IF doFrgVentilator THEN
    gStatusAnlage.Aktor[AKTOR_VENTILATOR] := STATUS_AKTIV;
ELSE
    gStatusAnlage.Aktor[AKTOR_VENTILATOR] := STATUS_NICHT_AKTIV;
END_IF;

aoFuVentilator := gAktoren.rVentilatorSollwert;

(*
===============================================================================
 LUFTAUFBEREITER
===============================================================================
 Direkte Ansteuerung
 Analoge Leistungsvorgabe analog zum Heizregister-Prinzip:
   - digitale Freigabe
   - analoger Sollwert
-------------------------------------------------------------------------------
*)

gStatusAnlage.LuftaufberTyp := gBetriebsparameter.Luftaufbereitung.Typ;


IF gAktoren.xFrgLuftaufbereiter THEN
    IF gAlarmBetriebLuftaufber THEN
        gStatusAnlage.Aktor[AKTOR_LUFTAUFBER] := STATUS_STOERUNG;
    ELSIF diBetriebLuftaufber THEN
        gStatusAnlage.Aktor[AKTOR_LUFTAUFBER] := STATUS_AKTIV;
    ELSE
        gStatusAnlage.Aktor[AKTOR_LUFTAUFBER] := STATUS_BEREIT;
    END_IF;
ELSE
    IF gAlarmBetriebLuftaufber THEN
        gStatusAnlage.Aktor[AKTOR_LUFTAUFBER] := STATUS_STOERUNG;
    ELSE
        gStatusAnlage.Aktor[AKTOR_LUFTAUFBER] := STATUS_NICHT_AKTIV;
    END_IF;
END_IF;

doFrgLuftaufber := gAktoren.xFrgLuftaufbereiter;
aoLeistVorgLuftaufber := gAktoren.rLuftaufbereiterSollwert;

(*
===============================================================================
 ABLUFTVENTILATOR
===============================================================================
 Direkte Ansteuerung
-------------------------------------------------------------------------------
*)

IF gAktoren.xFrgAbluftventilator THEN
    gStatusAnlage.Aktor[AKTOR_ABLUFTVENTILATOR] := STATUS_AKTIV;
ELSE
    gStatusAnlage.Aktor[AKTOR_ABLUFTVENTILATOR] := STATUS_NICHT_AKTIV;
END_IF;


doFrgAbluftventilator := gAktoren.xFrgAbluftventilator;
END_PROGRAM

PROGRAM HmiMappingCyclic
  VAR
    rt_Box_Aus : R_TRIG;
    rt_Box_Dauer : R_TRIG;
    rt_Box_Intervall : R_TRIG;
    rt_Box_Nachtr : R_TRIG;
    rt_Box_Stocktemp : R_TRIG;
    rt_Luftaufb_Auto : R_TRIG;
    rt_Luftaufb_Dauer : R_TRIG;
    rt_Luftaufb_Aus : R_TRIG;
    TOF_UmschBoxAktuell : TOF;  (* gemeinsam für Block A/B (schließen sich aus) *)
    TOF_UmschBox1 : TOF;  (* Block C (Einzelbox) *)
    xUmschSelAktuell : BOOL;
    xUmschSelBox1 : BOOL;
    lastBoxIndex : USINT;
    uIdx : USINT;
    firstStep : BOOL;
    xBox1BelegtLuefter : BOOL;
    xBox2BelegtLuefter : BOOL;
    TOF_Umsch : ARRAY[1..2] OF TOF;  (* eigener Hintergrund-Timer je Box *)
    xUmschTrig : ARRAY[1..2] OF BOOL;  (* Start-/Nachtrigger (Puls) je Box *)
    xZielAus : ARRAY[1..2] OF BOOL;  (* gewaehlte, noch nicht uebernommene Betriebsart *)
    xZielDauer : ARRAY[1..2] OF BOOL;
    xZielIntervall : ARRAY[1..2] OF BOOL;
    xZielNachtr : ARRAY[1..2] OF BOOL;
    xZielStocktemp : ARRAY[1..2] OF BOOL;
    xInitUmsch : BOOL := TRUE;
  END_VAR

(*
================================================================================
 File        : HMIMappingCyclic.st
 Project     : CControl_Lite
 Controller  : Schneider / EcoStruxure Machine Expert HVAC
 Author      : RIG Automation
 Created     : 2026-03-19
 Version     : V0.01
 Description :
    Zyklische Übergabe von Ein-/Ausgängen und aufbereiteten Messwerten an die HMI.

    Dieses Programm trennt bewusst zwischen:
      - Hardware-/Prozessabbild
      - interner Programmlogik
      - Visualisierungsdaten

    Die HMI liest ausschließlich die hier beschriebenen HMI-Variablen.
    Dadurch bleibt die Visualisierung von der eigentlichen I/O-Anbindung entkoppelt.

================================================================================
 Change History
--------------------------------------------------------------------------------
 Version | Date       | Author          | Description
--------------------------------------------------------------------------------
 V0.01   | 2026-03-19 | RIG Automation  | Initialerstellung HMI-Mapping für
                                        | digitale/analoge Ein- und Ausgänge
================================================================================
*)

(*
===============================================================================
 HMI-DATEN ZYKLISCH AKTUALISIEREN
-------------------------------------------------------------------------------
 Alle für die Visualisierung relevanten Ein- und Ausgangswerte werden in
 sprechende HMI-Variablen kopiert.
===============================================================================
*)
(*
---------------------------------------------------------------------------
Allgemein
---------------------------------------------------------------------------
*)
Konfig_SoftwareVersionPLC := gPlcSwVersion;
Konfig_idNameSteuerung := gPlcKonfigId;
gBetriebsparameter.Allgemein.StandortHoehe := Par_Anlage_Standorthoehe;


(*
---------------------------------------------------------------------------
Standard-Filterzeiten
---------------------------------------------------------------------------
*)
gBetriebsparameter.Sensoren.FilterzeitFrischluft := Sensoren_FilterzeitFrischluft;
gBetriebsparameter.Sensoren.FilterzeitAbluft := Sensoren_FilterzeitAbluft;
gBetriebsparameter.Sensoren.FilterzeitTrockenluft := Sensoren_FilterzeitTrockenluft;
gBetriebsparameter.Sensoren.FilterzeitStocktemp := Sensoren_FilterzeitStocktemp;

(*
---------------------------------------------------------------------------
Messbereiche Frischluft
---------------------------------------------------------------------------
*)
gBetriebsparameter.Sensoren.FrischlTempMessberMin := Sensoren_FrischlTempMessberMin;
gBetriebsparameter.Sensoren.FrischlTempMessberMax := Sensoren_FrischlTempMessberMax;
gBetriebsparameter.Sensoren.FrischlFeuchtMessberMin := Sensoren_FrischlFeuchteMessberMin;
gBetriebsparameter.Sensoren.FrischlFeuchtMessberMax := Sensoren_FrischlFeuchteMessberMax;

(*
---------------------------------------------------------------------------
Messbereiche Abluft
---------------------------------------------------------------------------
*)
gBetriebsparameter.Sensoren.AbluftTempMessberMin := Sensoren_AbluftTempMessberMin;
gBetriebsparameter.Sensoren.AbluftTempMessberMax := Sensoren_AbluftTempMessberMax;
gBetriebsparameter.Sensoren.AbluftFeuchtMessberMin := Sensoren_AbluftFeuchtMessberMin;
gBetriebsparameter.Sensoren.AbluftFeuchtMessberMax := Sensoren_AbluftFeuchtMessberMax;

(*
---------------------------------------------------------------------------
Messbereiche Trockenluft
---------------------------------------------------------------------------
*)
gBetriebsparameter.Sensoren.TrockenlTempMessberMin := Sensoren_TrockenlTempMessberMin;
gBetriebsparameter.Sensoren.TrockenlTempMessberMax := Sensoren_TrockenlTempMessberMax;
gBetriebsparameter.Sensoren.TrockenlFeuchtMessberMin := Sensoren_TrockenlFeuchtMessberMin;
gBetriebsparameter.Sensoren.TrockenlFeuchtMessberMax := Sensoren_TrockenlFeuchtMessberMax;

(*
---------------------------------------------------------------------------
Messbereiche Stocktemperatur
---------------------------------------------------------------------------
*)
gBetriebsparameter.Sensoren.StocktempMessberMin := Sensoren_StockTempMessberMin;
gBetriebsparameter.Sensoren.StocktempMessberMax := Sensoren_StockTempMessberMax;

(*
---------------------------------------------------------------------------
Sensor-Offsets
---------------------------------------------------------------------------
*)
gBetriebsparameter.Sensoren.OffsetFrischluftTemp := Sensoren_OffsetFrischluftTemp;
gBetriebsparameter.Sensoren.OffsetFrischluftFeuchte := Sensoren_OffsetFrischluftFeuchte;
gBetriebsparameter.Sensoren.OffsetAbluftBox1Temp := Sensoren_OffsetAbluftBox1Temp;
gBetriebsparameter.Sensoren.OffsetAbluftBox1Feuchte := Sensoren_OffsetAbluftBox1Feuchte;
gBetriebsparameter.Sensoren.OffsetAbluftBox2Temp := Sensoren_OffsetAbluftBox2Temp;
gBetriebsparameter.Sensoren.OffsetAbluftBox2Feuchte := Sensoren_OffsetAbluftBox2Feuchte;
gBetriebsparameter.Sensoren.OffsetTrockenluftTemp := Sensoren_OffsetTrockenluftTemp;
gBetriebsparameter.Sensoren.OffsetTrockenluftFeuchte := Sensoren_OffsetTrockenluftFeuchte;
gBetriebsparameter.Sensoren.OffsetStocktemp := Sensoren_OffsetStocktemp;

(*
---------------------------------------------------------------------------
Ausstattung / aktivierte Anlagenteile
---------------------------------------------------------------------------
Diese Werte sind vorläufige Defaultwerte und müssen später an die reale
Anlagenausstattung angepasst werden.
---------------------------------------------------------------------------
*)
gBetriebsparameter.Ausstattung.Box2 := Ausstattung_Box2;
gBetriebsparameter.Ausstattung.Abluftventilator := Ausstattung_Abluftventilator;
gBetriebsparameter.Ausstattung.SensorFrischluft := Ausstattung_SensorFrischluft;
gBetriebsparameter.Ausstattung.SensorAbluftBox1 := Ausstattung_SensorAbluftBox1;
gBetriebsparameter.Ausstattung.SensorAbluftBox2 := Ausstattung_SensorAbluftBox2;
gBetriebsparameter.Ausstattung.SensorTrockenluft := Ausstattung_SensorTrockenluft;
gBetriebsparameter.Ausstattung.SensorStocktemp := Ausstattung_SensorStocktemp;
gBetriebsparameter.Ausstattung.EndlagenVhdBoxenklappe1 := Ausstattung_EndlagenVhdBoxenklappe1;
gBetriebsparameter.Ausstattung.EndlagenVhdBoxenklappe2 := Ausstattung_EndlagenVhdBoxenklappe2;
gBetriebsparameter.Ausstattung.Luftaufbereiter := Ausstattung_Luftaufbereiter_Typ <> KEINER;

(*
---------------------------------------------------------------------------
Ventilator
---------------------------------------------------------------------------
*)
gBetriebsparameter.Ventilator.DrehzahlMin := Par_Ventilator_DrehzahlMin;
gBetriebsparameter.Ventilator.DrehzahlMax := Par_Ventilator_DrehzahlMax;
gBetriebsparameter.Ventilator.DrehzahlBeiAuskuehlphase := Par_Ventilator_DrehzahlBeiAuskuehlphase;
gBetriebsparameter.Ventilator.DrzUmschaltung := Par_Ventilator_DrzUmschaltung;
gBetriebsparameter.Ventilator.DrehzahlFixLuftaufbereiter := Par_Ventilator_DrehzahlFixLuftaufbereiter;
gBetriebsparameter.Ventilator.DrehzahlFixFrischluft := Par_Ventilator_DrehzahlFixFrischluft;
gBetriebsparameter.Ventilator.DrehzahlStrombegrenzung := Par_Ventilator_DrehzahlStrombegrenzung;
gBetriebsparameter.Ventilator.DrehzahlLeistungsreduziert := Par_Ventilator_DrehzahlLeistungsreduz;
gBetriebsparameter.Ventilator.ZeitRampeUp := Par_Ventilator_ZeitRampeUp;//[ms]
gBetriebsparameter.Ventilator.ZeitRampeDown := Par_Ventilator_ZeitRampeDown;//[ms]


(*
---------------------------------------------------------------------------
Luftaufbereitung
---------------------------------------------------------------------------
*)

//Allgemein
gBetriebsparameter.Luftaufbereitung.VerzWetterwechsel := Par_Luftaufbereitung_VerzWetterwechsel;
gBetriebsparameter.Luftaufbereitung.SaettigungFrischluftEin := Par_Luftaufbereitung_SaettigungFrischlEin;
gBetriebsparameter.Luftaufbereitung.Hysterese := Par_Luftaufbereitung_Hysterese;

//Betriebsarten
//--- Luftaufbereitung: Betriebsartenwahl (flankengesteuert, gegenseitig verriegelt) ---
rt_Luftaufb_Auto (CLK := Par_Luftaufbereitung_AutomatikbetriebEin);
rt_Luftaufb_Dauer(CLK := Par_Luftaufbereitung_DauerbetriebEin);
rt_Luftaufb_Aus  (CLK := Par_Luftaufbereitung_Aus);

IF rt_Luftaufb_Auto.Q THEN
	Par_Luftaufbereitung_DauerbetriebEin     := FALSE;
	Par_Luftaufbereitung_Aus                 := FALSE;
ELSIF rt_Luftaufb_Dauer.Q THEN
	Par_Luftaufbereitung_AutomatikbetriebEin := FALSE;
	Par_Luftaufbereitung_Aus                 := FALSE;
ELSIF rt_Luftaufb_Aus.Q THEN
	Par_Luftaufbereitung_AutomatikbetriebEin := FALSE;
	Par_Luftaufbereitung_DauerbetriebEin     := FALSE;
END_IF;

//Aufbereitete Anwahl an interne Betriebsparameter uebergeben
gBetriebsparameter.Luftaufbereitung.AutomatikbetriebEin := Par_Luftaufbereitung_AutomatikbetriebEin;
gBetriebsparameter.Luftaufbereitung.DauerbetriebEin     := Par_Luftaufbereitung_DauerbetriebEin;
gBetriebsparameter.Luftaufbereitung.Aus                 := Par_Luftaufbereitung_Aus;

//Spezifisch Heizregister
gBetriebsparameter.Luftaufbereitung.P := Par_Luftaufbereitung_P;
gBetriebsparameter.Luftaufbereitung.I := Par_Luftaufbereitung_I;
gBetriebsparameter.Luftaufbereitung.D := Par_Luftaufbereitung_D;
gBetriebsparameter.Luftaufbereitung.DrehzahlVorgabeMin := Par_Luftaufbereitung_DrehzahlVorgabeMin;
gBetriebsparameter.Luftaufbereitung.DrehzahlVorgabeMax := Par_Luftaufbereitung_DrehzahlVorgabeMax;
gBetriebsparameter.Luftaufbereitung.TempVorgabeSoll := Par_Luftaufbereitung_TempVorgabeSoll;
//Spezifisch Ofen
gBetriebsparameter.Luftaufbereitung.VerzBetriebsmeldung := Par_Luftaufbereitung_VerzBetriebsmeldung;
gBetriebsparameter.Luftaufbereitung.Auskuehlzeit := Par_Luftaufbereitung_Auskuehlzeit;
gBetriebsparameter.Luftaufbereitung.BetriebsmeldungVorh := Par_Luftaufbereitung_BetriebsmeldungVorh;

(*
---------------------------------------------------------------------------
Abluft
---------------------------------------------------------------------------
*)
gBetriebsparameter.Abluftventilator.FeuchteSoll := Par_Abluft_FeuchteSoll;
gBetriebsparameter.Abluftventilator.Hysterese := Par_Abluft_FeuchteHysterese;

(*
---------------------------------------------------------------------------
Schlechtwetter
---------------------------------------------------------------------------
*)

//======== Box 1 =========

//Sensortype 
gBetriebsparameter.SchlechtwetterBoxen[1].AuswahlSensorGrenzwert := Par_Schlechtwetter_Box1_Sensortype;
//Feuchte
gBetriebsparameter.SchlechtwetterBoxen[1].Stufe[1].MaterialfeuchteStufe := Par_Schlechtwetter_Box1_MaterialfeuchteStufe1;
gBetriebsparameter.SchlechtwetterBoxen[1].Stufe[2].MaterialfeuchteStufe := Par_Schlechtwetter_Box1_MaterialfeuchteStufe2;
gBetriebsparameter.SchlechtwetterBoxen[1].Stufe[3].MaterialfeuchteStufe := Par_Schlechtwetter_Box1_MaterialfeuchteStufe3;
gBetriebsparameter.SchlechtwetterBoxen[1].Stufe[4].MaterialfeuchteStufe := Par_Schlechtwetter_Box1_MaterialfeuchteStufe4;
gBetriebsparameter.SchlechtwetterBoxen[1].Stufe[5].MaterialfeuchteStufe := Par_Schlechtwetter_Box1_MaterialfeuchteStufe5;
gBetriebsparameter.SchlechtwetterBoxen[1].Stufe[6].MaterialfeuchteStufe := Par_Schlechtwetter_Box1_MaterialfeuchteStufe6;
//Saettigung
gBetriebsparameter.SchlechtwetterBoxen[1].Stufe[1].Saettigungsdefizit := Par_Schlechtwetter_Box1_Saettigungsdefizit1;
gBetriebsparameter.SchlechtwetterBoxen[1].Stufe[2].Saettigungsdefizit := Par_Schlechtwetter_Box1_Saettigungsdefizit2;
gBetriebsparameter.SchlechtwetterBoxen[1].Stufe[3].Saettigungsdefizit := Par_Schlechtwetter_Box1_Saettigungsdefizit3;
gBetriebsparameter.SchlechtwetterBoxen[1].Stufe[4].Saettigungsdefizit := Par_Schlechtwetter_Box1_Saettigungsdefizit4;
gBetriebsparameter.SchlechtwetterBoxen[1].Stufe[5].Saettigungsdefizit := Par_Schlechtwetter_Box1_Saettigungsdefizit5;
gBetriebsparameter.SchlechtwetterBoxen[1].Stufe[6].Saettigungsdefizit := Par_Schlechtwetter_Box1_Saettigungsdefizit6;
// Zeit Lauf
gBetriebsparameter.SchlechtwetterBoxen[1].Stufe[1].SchlechtwetterZeitLauf := Par_Schlechtwetter_Box1_ZeitLauf1;
gBetriebsparameter.SchlechtwetterBoxen[1].Stufe[2].SchlechtwetterZeitLauf := Par_Schlechtwetter_Box1_ZeitLauf2;
gBetriebsparameter.SchlechtwetterBoxen[1].Stufe[3].SchlechtwetterZeitLauf := Par_Schlechtwetter_Box1_ZeitLauf3;
gBetriebsparameter.SchlechtwetterBoxen[1].Stufe[4].SchlechtwetterZeitLauf := Par_Schlechtwetter_Box1_ZeitLauf4;
gBetriebsparameter.SchlechtwetterBoxen[1].Stufe[5].SchlechtwetterZeitLauf := Par_Schlechtwetter_Box1_ZeitLauf5;
gBetriebsparameter.SchlechtwetterBoxen[1].Stufe[6].SchlechtwetterZeitLauf := Par_Schlechtwetter_Box1_ZeitLauf6;
// Zeit Pause
gBetriebsparameter.SchlechtwetterBoxen[1].Stufe[1].SchlechtwetterZeitPause := Par_Schlechtwetter_Box1_ZeitPause1;
gBetriebsparameter.SchlechtwetterBoxen[1].Stufe[2].SchlechtwetterZeitPause := Par_Schlechtwetter_Box1_ZeitPause2;
gBetriebsparameter.SchlechtwetterBoxen[1].Stufe[3].SchlechtwetterZeitPause := Par_Schlechtwetter_Box1_ZeitPause3;
gBetriebsparameter.SchlechtwetterBoxen[1].Stufe[4].SchlechtwetterZeitPause := Par_Schlechtwetter_Box1_ZeitPause4;
gBetriebsparameter.SchlechtwetterBoxen[1].Stufe[5].SchlechtwetterZeitPause := Par_Schlechtwetter_Box1_ZeitPause5;
gBetriebsparameter.SchlechtwetterBoxen[1].Stufe[6].SchlechtwetterZeitPause := Par_Schlechtwetter_Box1_ZeitPause6;

gBetriebsparameter.SchlechtwetterBoxen[1].MaterialfeuchteIst := gBetriebsparameter.Boxen[1].AktuelleTrockengutFeuchte;
gBetriebsparameter.SchlechtwetterBoxen[1].HystereseGrenzwert := gBetriebsparameter.Luftaufbereitung.Hysterese;

//======== Box 2 =========

//Sensortype 
gBetriebsparameter.SchlechtwetterBoxen[2].AuswahlSensorGrenzwert := Par_Schlechtwetter_Box2_Sensortype;
//Feuchte
gBetriebsparameter.SchlechtwetterBoxen[2].Stufe[1].MaterialfeuchteStufe := Par_Schlechtwetter_Box2_MaterialfeuchteStufe1;
gBetriebsparameter.SchlechtwetterBoxen[2].Stufe[2].MaterialfeuchteStufe := Par_Schlechtwetter_Box2_MaterialfeuchteStufe2;
gBetriebsparameter.SchlechtwetterBoxen[2].Stufe[3].MaterialfeuchteStufe := Par_Schlechtwetter_Box2_MaterialfeuchteStufe3;
gBetriebsparameter.SchlechtwetterBoxen[2].Stufe[4].MaterialfeuchteStufe := Par_Schlechtwetter_Box2_MaterialfeuchteStufe4;
gBetriebsparameter.SchlechtwetterBoxen[2].Stufe[5].MaterialfeuchteStufe := Par_Schlechtwetter_Box2_MaterialfeuchteStufe5;
gBetriebsparameter.SchlechtwetterBoxen[2].Stufe[6].MaterialfeuchteStufe := Par_Schlechtwetter_Box2_MaterialfeuchteStufe6;
//Saettigung
gBetriebsparameter.SchlechtwetterBoxen[2].Stufe[1].Saettigungsdefizit := Par_Schlechtwetter_Box2_Saettigungsdefizit1;
gBetriebsparameter.SchlechtwetterBoxen[2].Stufe[2].Saettigungsdefizit := Par_Schlechtwetter_Box2_Saettigungsdefizit2;
gBetriebsparameter.SchlechtwetterBoxen[2].Stufe[3].Saettigungsdefizit := Par_Schlechtwetter_Box2_Saettigungsdefizit3;
gBetriebsparameter.SchlechtwetterBoxen[2].Stufe[4].Saettigungsdefizit := Par_Schlechtwetter_Box2_Saettigungsdefizit4;
gBetriebsparameter.SchlechtwetterBoxen[2].Stufe[5].Saettigungsdefizit := Par_Schlechtwetter_Box2_Saettigungsdefizit5;
gBetriebsparameter.SchlechtwetterBoxen[2].Stufe[6].Saettigungsdefizit := Par_Schlechtwetter_Box2_Saettigungsdefizit6;
// Zeit Lauf
gBetriebsparameter.SchlechtwetterBoxen[2].Stufe[1].SchlechtwetterZeitLauf := Par_Schlechtwetter_Box2_ZeitLauf1;
gBetriebsparameter.SchlechtwetterBoxen[2].Stufe[2].SchlechtwetterZeitLauf := Par_Schlechtwetter_Box2_ZeitLauf2;
gBetriebsparameter.SchlechtwetterBoxen[2].Stufe[3].SchlechtwetterZeitLauf := Par_Schlechtwetter_Box2_ZeitLauf3;
gBetriebsparameter.SchlechtwetterBoxen[2].Stufe[4].SchlechtwetterZeitLauf := Par_Schlechtwetter_Box2_ZeitLauf4;
gBetriebsparameter.SchlechtwetterBoxen[2].Stufe[5].SchlechtwetterZeitLauf := Par_Schlechtwetter_Box2_ZeitLauf5;
gBetriebsparameter.SchlechtwetterBoxen[2].Stufe[6].SchlechtwetterZeitLauf := Par_Schlechtwetter_Box2_ZeitLauf6;
// Zeit Pause
gBetriebsparameter.SchlechtwetterBoxen[2].Stufe[1].SchlechtwetterZeitPause := Par_Schlechtwetter_Box2_ZeitPause1;
gBetriebsparameter.SchlechtwetterBoxen[2].Stufe[2].SchlechtwetterZeitPause := Par_Schlechtwetter_Box2_ZeitPause2;
gBetriebsparameter.SchlechtwetterBoxen[2].Stufe[3].SchlechtwetterZeitPause := Par_Schlechtwetter_Box2_ZeitPause3;
gBetriebsparameter.SchlechtwetterBoxen[2].Stufe[4].SchlechtwetterZeitPause := Par_Schlechtwetter_Box2_ZeitPause4;
gBetriebsparameter.SchlechtwetterBoxen[2].Stufe[5].SchlechtwetterZeitPause := Par_Schlechtwetter_Box2_ZeitPause5;
gBetriebsparameter.SchlechtwetterBoxen[2].Stufe[6].SchlechtwetterZeitPause := Par_Schlechtwetter_Box2_ZeitPause6;

gBetriebsparameter.SchlechtwetterBoxen[2].MaterialfeuchteIst := gBetriebsparameter.Boxen[2].AktuelleTrockengutFeuchte;
gBetriebsparameter.SchlechtwetterBoxen[2].HystereseGrenzwert := gBetriebsparameter.Luftaufbereitung.Hysterese;

(*
---------------------------------------------------------------------------
Klappen/Boxen
---------------------------------------------------------------------------
*)
gBetriebsparameter.KlappenBoxen[1].Laufzeit := Klappen_Boxen_Box1_Laufzeit;
gBetriebsparameter.KlappenBoxen[2].Laufzeit := Klappen_Boxen_Box2_Laufzeit;

(*
---------------------------------------------------------------------------
Luftaufbereitung Allgemein
---------------------------------------------------------------------------
*)
gBetriebsparameter.Luftaufbereitung.Typ := Ausstattung_Luftaufbereiter_Typ;

(*
---------------------------------------------------------------------------
Strombegrenzung
---------------------------------------------------------------------------
*)
gBetriebsparameter.Strombegrenzung.StartStd := Par_Strombegrenzung_StartMin;
gBetriebsparameter.Strombegrenzung.StartMin := Par_Strombegrenzung_StartStd;
gBetriebsparameter.Strombegrenzung.StoppStd := Par_Strombegrenzung_StoppMin;
gBetriebsparameter.Strombegrenzung.StoppMin := Par_Strombegrenzung_StoppStd;
(*
---------------------------------------------------------------------------
Tarifabschaltung
---------------------------------------------------------------------------
*)
gBetriebsparameter.Tarifabschaltung.Zeitfenster.StartStd := Par_Tarifabschaltung_Start_Std;
gBetriebsparameter.Tarifabschaltung.Zeitfenster.StartMin := Par_Tarifabschaltung_Start_Min;
gBetriebsparameter.Tarifabschaltung.Zeitfenster.StoppStd := Par_Tarifabschaltung_Stopp_Std;
gBetriebsparameter.Tarifabschaltung.Zeitfenster.StoppMin := Par_Tarifabschaltung_Stopp_Min;
gBetriebsparameter.Tarifabschaltung.VorlaufzeitAbschaltungLuftaufb := Par_Vorlaufzeit_Luftaufb_Tarifabschalt;

(*
---------------------------------------------------------------------------
Verzoegerungen (alle in ms) 
---------------------------------------------------------------------------
*)
gBetriebsparameter.Verzoegerungen.Fehler                    := Par_Verz_Fehler;
gBetriebsparameter.Verzoegerungen.Warnungen                 := Par_Verz_Warnungen;
gBetriebsparameter.Verzoegerungen.AenderungKlappenstellung  := Par_Verz_Aenderung_Klappenstellung;
gBetriebsparameter.Verzoegerungen.UmschaltungBetriebsartBox := Par_Verz_Umsch_Betriebsart_Box;


(*
-------------------------------------------------------------------------------
 Betriebsart / allgemeiner Zustand
-------------------------------------------------------------------------------
*)
HMI_TEST_diIoTestAktiv:= (gAktModus = IOTEST);

(*
-------------------------------------------------------------------------------
 Digitale Eingänge an HMI übergeben
-------------------------------------------------------------------------------
*)
HMI_IN_diBox1Offen  		:= diBox1Offen;
HMI_IN_diBox1Geschl  		:= diBox1Geschl;
HMI_IN_diBox2Offen  		:= diBox2Offen;
HMI_IN_diBox2Geschl 		:= diBox2Geschl;
HMI_IN_diBetriebLuftaufber 	:= diBetriebLuftaufber;
HMI_IN_diBetriebVentilator 	:= diBetriebVentilator;

(*
-------------------------------------------------------------------------------
 Analoge Eingänge an HMI übergeben
-------------------------------------------------------------------------------
 Es werden bereits skalierte Engineering-Werte an die HMI übergeben.
-------------------------------------------------------------------------------
*)
HMI_IN_aiFrischluftTemp       := gStatusAnlage.FrischluftTemperatur;
HMI_IN_aiFrischluftFeuchte    := gStatusAnlage.FrischluftFeuchte;
HMI_IN_aiAbluftBox1Temp       := gStatusAnlage.AbluftBox1Temp;
HMI_IN_aiAbluftBox1Feuchte    := gStatusAnlage.AbluftBox1Feuchte;
HMI_IN_aiTrockenluftTemp      := gStatusAnlage.TrockenluftTemperatur;
HMI_IN_aiTrockenluftFeuchte   := gStatusAnlage.TrockenluftFeuchte;
HMI_IN_aiAbluftBox2Temp       := gStatusAnlage.AbluftBox2Temp;
HMI_IN_aiAbluftBox2Feuchte    := gStatusAnlage.AbluftBox2Feuchte;
HMI_IN_aiStocktemp            := gStatusAnlage.StockTemperatur;


(*
-------------------------------------------------------------------------------
 Digitale Ausgänge an HMI übergeben
-------------------------------------------------------------------------------
 Hier werden die internen Soll-/Freigabesignale visualisiert.
-------------------------------------------------------------------------------
*)
HMI_IN_doFrgLuftaufber     		:= doFrgLuftaufber;
HMI_IN_doFrgBox1            	:= doFrgBox1;
HMI_IN_doFrgBox2           		:= doFrgBox2;
HMI_IN_doFrgAbluftvent	     	:= doFrgAbluftventilator;
HMI_IN_doFrgVentilator	     	:= doFrgVentilator;

(*
-------------------------------------------------------------------------------
 Analogausgänge an HMI übergeben
-------------------------------------------------------------------------------
 Die HMI erhält die Engineering-Sollwerte sowie optional die bereits
 skalierten Hardwarewerte.
-------------------------------------------------------------------------------
*)
HMI_IN_aoFuVentilator   	  := aoFuVentilator;
HMI_IN_aoLeistVorgLuftaufber  := aoLeistVorgLuftaufber;


(*
-------------------------------------------------------------------------------
 Berechnete Werte an HMI übergeben
-------------------------------------------------------------------------------
*)
HMI_IN_FrischlSaettigunsDefizit := gStatusAnlage.FrischluftSaettDefizit;
HMI_IN_TrockenluftSaettigunsDefizit := gStatusAnlage.TrockenluftSaettDefizit;

(*
-------------------------------------------------------------------------------
 I/O-Testdaten an HMI übergeben
-------------------------------------------------------------------------------
 So sieht man in der Visu sofort, ob Testbetrieb aktiv ist und welche
 Testwerte gerade anliegen.
-------------------------------------------------------------------------------
*)


(* PLC OUT - HMI IN *)

//digital
HMI_TEST_diBox1Offen     		:= gIoTest.DigitalIn.diBox1Offen;
HMI_TEST_diBox1Geschl  	 		:= gIoTest.DigitalIn.diBox1Geschl;
HMI_TEST_diBox2Offen   		 	:= gIoTest.DigitalIn.diBox2Offen;
HMI_TEST_diBox2Geschl    		:= gIoTest.DigitalIn.diBox2Geschl;
HMI_TEST_diBetriebLuftaufber  	:= gIoTest.DigitalIn.diBetriebLuftaufber;
HMI_TEST_diBetriebVentilator 	:= gIoTest.DigitalIn.diBetriebVentilator;

//analog
HMI_TEST_aiFrischluftTemp  		:= gIoTest.AnalogIn.aiFrischluftTemp;
HMI_TEST_aiFrischluftFeuchte  	:= gIoTest.AnalogIn.aiFrischluftFeuchte;
HMI_TEST_aiAbluftBox1Temp     	:= gIoTest.AnalogIn.aiAbluftBox1Temp;
HMI_TEST_aiAbluftBox1Feuchte  	:= gIoTest.AnalogIn.aiAbluftBox1Feucht;
HMI_TEST_aiTrockenluftTemp 	  	:= gIoTest.AnalogIn.aiTrockenluftTemp;
HMI_TEST_aiTrockenluftFeuchte 	:= gIoTest.AnalogIn.aiTrockenluftFeucht;
HMI_TEST_aiAbluftBox2Temp  	  	:= gIoTest.AnalogIn.aiAbluftBox2Temp;
HMI_TEST_aiAbluftBox2Feuchte  	:= gIoTest.AnalogIn.aiAbluftBox2Feucht;
HMI_TEST_aiStocktemp   		  	:= gIoTest.AnalogIn.aiStocktemp;

(* HMI IN - PLC OUT *)

//digital
gIoTest.DigitalOut.doFrgLuftaufber			:= HMI_TEST_doFrgLuftaufber;
gIoTest.DigitalOut.doFrgBox1				:= HMI_TEST_doFrgBox1;
gIoTest.DigitalOut.doFrgBox2				:= HMI_TEST_doFrgBox2;
gIoTest.DigitalOut.doFrgAbluftventilator	:= HMI_TEST_doFrgAbluftventilator;
gIoTest.DigitalOut.doFrgVentilator			:= HMI_TEST_doFrgVentilator;

//analog
gIoTest.AnalogOut.aoFuVentilator			:= HMI_TEST_aoFuVentilator;
gIoTest.AnalogOut.aoLeistVorgLuftaufber 	:= HMI_TEST_aoLeistVorgLuftaufber;



(*
-------------------------------------------------------------------------------
 IO-MAPPING BOXEN 
-------------------------------------------------------------------------------
 Hier werden die Daten der Detailansichten der Boxen auf das allgemeine 
 PopUp geschrieben. Das allgemeine PopUp wird immer angezeigt wenn auf eine
 der Boxen geklickt wird. Die Daten der jeweiligen Box die ausgewählt wurde 
 werden dann auf dieses PopUp gemappet.
-------------------------------------------------------------------------------
*)

//======== Allgemein =========

gBetriebsparameter.Boxen[1].NameBox := Par_Box1_Name;
gBetriebsparameter.Boxen[2].NameBox := Par_Box2_Name;

//Trockengut
gBetriebsparameter.Boxen[1].Trockengut := Par_Boxen_1_Trockengut;
gBetriebsparameter.Boxen[2].Trockengut := Par_Boxen_2_Trockengut;

//Einstellung und Konfiguration Stellung Klappen
gBetriebsparameter.Boxen[1].StellungKlappe1 := Par_Box1_StellungKlappe1;
gBetriebsparameter.Boxen[1].StellungKlappe2 := Par_Box1_StellungKlappe2;
gBetriebsparameter.Boxen[2].StellungKlappe1 := Par_Box2_StellungKlappe1;
gBetriebsparameter.Boxen[2].StellungKlappe2 := Par_Box2_StellungKlappe2;

//Stocktemperatur
gBetriebsparameter.Boxen[1].StocktemperaturHysterese := Par_Stocktemperatur_Box1_Hysterese;
gBetriebsparameter.Boxen[2].StocktemperaturHysterese := Par_Stocktemperatur_Box2_Hysterese;

(*
-------------------------------------------------------------------------------
 Verriegelung Box-Betriebsarten (1 Luefter -> nur eine Box gleichzeitig)
 Belegt eine Box den Luefter durchgehend, wird bei der anderen Box
 Dauer-/Intervallbetrieb gesperrt (nur HMI-Hinweis).
-------------------------------------------------------------------------------
*)
// Reset
gStatusAnlage.Box[1].SperreDauerbetrieb     := FALSE;
gStatusAnlage.Box[1].SperreIntervallbetrieb := FALSE;
gStatusAnlage.Box[2].SperreDauerbetrieb     := FALSE;
gStatusAnlage.Box[2].SperreIntervallbetrieb := FALSE;

IF gBetriebsparameter.Ausstattung.Box2 THEN

    // "belegt den Luefter durchgehend" = Dauerbetrieb oder Stocktemperatur
    xBox1BelegtLuefter := gBetriebsparameter.Boxen[1].DauerbetriebEin
                          OR gBetriebsparameter.Boxen[1].StocktemperaturEin;
    xBox2BelegtLuefter := gBetriebsparameter.Boxen[2].DauerbetriebEin
                          OR gBetriebsparameter.Boxen[2].StocktemperaturEin;

    // Box 2 belegt den Luefter -> Box 1 sperren
    IF xBox2BelegtLuefter THEN
        gStatusAnlage.Box[1].SperreDauerbetrieb     := TRUE;
        gStatusAnlage.Box[1].SperreIntervallbetrieb := TRUE;
    ELSIF gBetriebsparameter.Boxen[2].IntervallbetriebEin THEN
        // Intervall der einen Box -> Dauerbetrieb der anderen wuerde stoeren
        gStatusAnlage.Box[1].SperreDauerbetrieb     := TRUE;
    END_IF;

    // Box 1 belegt den Luefter -> Box 2 sperren
    IF xBox1BelegtLuefter THEN
        gStatusAnlage.Box[2].SperreDauerbetrieb     := TRUE;
        gStatusAnlage.Box[2].SperreIntervallbetrieb := TRUE;
    ELSIF gBetriebsparameter.Boxen[1].IntervallbetriebEin THEN
        gStatusAnlage.Box[2].SperreDauerbetrieb     := TRUE;
    END_IF;

END_IF;

// --- HMI-Spiegel ---
HMI_IN_Box1_SperreDauerbetrieb     := gStatusAnlage.Box[1].SperreDauerbetrieb;
HMI_IN_Box1_SperreIntervallbetrieb := gStatusAnlage.Box[1].SperreIntervallbetrieb;
HMI_IN_Box2_SperreDauerbetrieb     := gStatusAnlage.Box[2].SperreDauerbetrieb;
HMI_IN_Box2_SperreIntervallbetrieb := gStatusAnlage.Box[2].SperreIntervallbetrieb;

// Aktuell-PopUp je nach angezeigter Box
IF HMI_OUT_Box_Aktuell_BoxIndex = BOX_2 THEN
    HMI_IN_Box_Aktuell_SperreDauerbetrieb     := gStatusAnlage.Box[2].SperreDauerbetrieb;
    HMI_IN_Box_Aktuell_SperreIntervallbetrieb := gStatusAnlage.Box[2].SperreIntervallbetrieb;
ELSE
    HMI_IN_Box_Aktuell_SperreDauerbetrieb     := gStatusAnlage.Box[1].SperreDauerbetrieb;
    HMI_IN_Box_Aktuell_SperreIntervallbetrieb := gStatusAnlage.Box[1].SperreIntervallbetrieb;
END_IF;

//======== Box 1 =========
HMI_IN_Box1_IconWitterung := gStatusAnlage.Box[1].IconWitterung;
HMI_IN_Box1_LaufRestzeitMinuten := gStatusAnlage.Box[1].LaufRestzeitMinuten;
HMI_IN_Box1_LaufRestzeitStunden := gStatusAnlage.Box[1].LaufRestzeitStunden;
HMI_IN_Box1_Status := TO_UINT(gStatusAnlage.Box[1].Status);
HMI_IN_Box1_TextIndexLaufzeit := gStatusAnlage.Box[1].TextIndexLaufzeit;
HMI_IN_Box1_TrockengutIcon := gStatusAnlage.Box[1].TrockengutIcon;
HMI_IN_Box1_AnzeigeLaufRestzeit := gStatusAnlage.Box[1].AnzeigeLaufRestzeit;

//TODO RIG: Noch zu verschalten
//HMI_IN_Box1_RestzeitUmschVerzBetriebsart

//======== Box 2 =========
HMI_IN_Box2_IconWitterung := gStatusAnlage.Box[2].IconWitterung;
HMI_IN_Box2_LaufRestzeitMinuten := gStatusAnlage.Box[2].LaufRestzeitMinuten;
HMI_IN_Box2_LaufRestzeitStunden := gStatusAnlage.Box[2].LaufRestzeitStunden;
HMI_IN_Box2_Status := TO_UINT(gStatusAnlage.Box[2].Status);
HMI_IN_Box2_TextIndexLaufzeit := gStatusAnlage.Box[2].TextIndexLaufzeit;
HMI_IN_Box2_TrockengutIcon := gStatusAnlage.Box[2].TrockengutIcon;
HMI_IN_Box2_AnzeigeLaufRestzeit := gStatusAnlage.Box[2].AnzeigeLaufRestzeit;

//TODO RIG: Noch zu verschalten
//HMI_IN_Box2_RestzeitUmschVerzBetriebsart

IF lastBoxIndex <> HMI_OUT_Box_Aktuell_BoxIndex THEN
	firstStep := TRUE;
	lastBoxIndex := HMI_OUT_Box_Aktuell_BoxIndex;
END_IF;

(*
-------------------------------------------------------------------------------
 Zusatzmeldung Anlagenstatus (vereinfacht fuer Lite) - nur Statustext
-------------------------------------------------------------------------------
*)
IF gAktModus = STILLSTAND THEN
    IF gAktoren.xLuftaufbNachlauf AND NOT gAktoren.xFrgLuftaufbereiter THEN
        HMI_Zusatzmeldung_Statustext := ZM_AUSKUEHLZEIT_WLO_AKTIV;      // Auskuehlung laeuft
    ELSIF gCmdAnlage.FehlerStopp THEN
        HMI_Zusatzmeldung_Statustext := ZM_STILLSTAND_FEHLERSTOPP;      // Fehler - kein Start
    ELSE
        HMI_Zusatzmeldung_Statustext := ZM_STILLSTAND_BEREIT;          // bereit
    END_IF;

ELSIF gAktModus = IOTEST THEN
    HMI_Zusatzmeldung_Statustext := ZM_STILLSTAND_IOTEST_NICHT_ABGE;    // I/O-Test aktiv

ELSE   // BETRIEB
    HMI_Zusatzmeldung_Restzeit 	:= 0;   //Kein Countdown
    HMI_Zusatzmeldung_Sanduhr 	:= 0;	//Keine Sanduhr
    IF gCmdAnlage.xTarifAbschaltung THEN
        HMI_Zusatzmeldung_Statustext := ZM_TARIFABSCHALTUNG_AKTIV;
    ELSIF gCmdAnlage.xTarifAbschaltungLuftaufb THEN
        HMI_Zusatzmeldung_Statustext := ZM_FRISCHLUFTB_VLZ_TARIF;
    ELSIF Strombegrenzung.StrombegrenzungEin THEN
        HMI_Zusatzmeldung_Statustext := ZM_STROMBEGRENZUNG_AKTIV;
    ELSIF (gStatusAnlage.Aktor[AKTOR_KLAPPE_BOX_1] = STATUS_IN_BEWEGUNG)
       OR (gStatusAnlage.Aktor[AKTOR_KLAPPE_BOX_2] = STATUS_IN_BEWEGUNG) THEN
        HMI_Zusatzmeldung_Statustext := ZM_KLAPPEN_WERDEN_UMGESCHALTET;
        HMI_Zusatzmeldung_Restzeit   := HMI_IN_Box_Aktuell_RestzeitUmschVerzBetriebsart;  
        HMI_Zusatzmeldung_Sanduhr := 1;
    ELSIF gAktoren.xLuftaufbNachlauf AND NOT gAktoren.xFrgLuftaufbereiter THEN
        HMI_Zusatzmeldung_Statustext := ZM_AUSKUEHLZEIT_WLO_AKTIV;
        HMI_Zusatzmeldung_Restzeit   := gAktoren.uRestAuskuehlzeitLuftaufb;   
    ELSE
        HMI_Zusatzmeldung_Statustext := ZM_FRISCHLUFTBETRIEB;
    END_IF;
END_IF;


//Box 1 auf Aktualfenster PopUp schreiben
IF HMI_OUT_Box_Aktuell_BoxIndex = BOX_1 THEN
	
	IF firstStep THEN
		HMI_OUT_Box_Aktuell_Aus                 := xZielAus[1];
		HMI_OUT_Box_Aktuell_DauerbetriebEin     := xZielDauer[1];
		HMI_OUT_Box_Aktuell_IntervallbetriebEIn := xZielIntervall[1];
		HMI_OUT_Box_Aktuell_NachtrocknungEin    := xZielNachtr[1];
		HMI_OUT_Box_Aktuell_StocktemperaturEin  := xZielStocktemp[1];
		HMI_OUT_Box_Aktuell_TrockengutfeuchteAktuell := gBetriebsparameter.Boxen[1].AktuelleTrockengutFeuchte;
		HMI_OUT_Box_Aktuell_StocktemperaturSoll := gBetriebsparameter.Boxen[1].StocktemperaturSoll;
		firstStep := FALSE;
	END_IF;
		
	//--- Gewaehlte Betriebsart als Ziel merken + Hintergrund-Timer starten ---
	IF rt_Box_Aus.Q OR rt_Box_Dauer.Q OR rt_Box_Intervall.Q OR rt_Box_Nachtr.Q OR rt_Box_Stocktemp.Q THEN
		xZielAus[1]       := HMI_OUT_Box_Aktuell_Aus;
		xZielDauer[1]     := HMI_OUT_Box_Aktuell_DauerbetriebEin;
		xZielIntervall[1] := HMI_OUT_Box_Aktuell_IntervallbetriebEIn;
		xZielNachtr[1]    := HMI_OUT_Box_Aktuell_NachtrocknungEin;
		xZielStocktemp[1] := HMI_OUT_Box_Aktuell_StocktemperaturEin;
		xUmschTrig[1]     := TRUE;
	END_IF;
	
	HMI_IN_Box_Aktuell_RestzeitUmschVerzBetriebsart := TO_UINT(gBetriebsparameter.Verzoegerungen.UmschaltungBetriebsartBox - TOF_Umsch[1].ET);
	//Aktuelle Trockengutfeuchte - Einstellung aus HMI
	gBetriebsparameter.Boxen[1].AktuelleTrockengutFeuchte := HMI_OUT_Box_Aktuell_TrockengutfeuchteAktuell;
	gBetriebsparameter.Boxen[1].StocktemperaturSoll := 	HMI_OUT_Box_Aktuell_StocktemperaturSoll;
	
	
	//PLC -> HMI
	HMI_IN_Box_Aktuell_Name := gBetriebsparameter.Boxen[1].NameBox;
	HMI_IN_Box_Aktuell_Temp := gStatusAnlage.AbluftBox1Temp;
	HMI_IN_Box_Aktuell_Feucht := gStatusAnlage.AbluftBox1Feuchte;	
	HMI_IN_Box_Aktuell_TrockengutIcon := gStatusAnlage.Box[1].TrockengutIcon;
	HMI_IN_Box_Aktuell_LaufRestzeitMinuten := gStatusAnlage.Box[1].LaufRestzeitMinuten;
	HMI_IN_Box_Aktuell_LaufRestzeitStunden := gStatusAnlage.Box[1].LaufRestzeitStunden;
	HMI_IN_Box_Aktuell_IconWitterung := gStatusAnlage.Box[1].IconWitterung;
	HMI_IN_Box_Aktuell_Status := TO_INT(gStatusAnlage.Box[1].Status);
	HMI_IN_Box_Aktuell_TextIndexLaufzeit := gStatusAnlage.Box[1].TextIndexLaufzeit;
	HMI_IN_Box_Aktuell_AnzeigeLaufRestzeit := gStatusAnlage.Box[1].AnzeigeLaufRestzeit;
	
	
//Box 2 auf Aktualfenster-PopUp schreiben
ELSIF HMI_OUT_Box_Aktuell_BoxIndex = BOX_2 THEN

	IF firstStep THEN
		HMI_OUT_Box_Aktuell_Aus                 := xZielAus[2];
		HMI_OUT_Box_Aktuell_DauerbetriebEin     := xZielDauer[2];
		HMI_OUT_Box_Aktuell_IntervallbetriebEIn := xZielIntervall[2];
		HMI_OUT_Box_Aktuell_NachtrocknungEin    := xZielNachtr[2];
		HMI_OUT_Box_Aktuell_StocktemperaturEin  := xZielStocktemp[2];
		HMI_OUT_Box_Aktuell_TrockengutfeuchteAktuell := gBetriebsparameter.Boxen[2].AktuelleTrockengutFeuchte;
		HMI_OUT_Box_Aktuell_StocktemperaturSoll := gBetriebsparameter.Boxen[2].StocktemperaturSoll;
		firstStep := FALSE;
	END_IF;

	//HMI -> PLC	
	//--- Gewaehlte Betriebsart als Ziel merken + Hintergrund-Timer starten ---
	IF rt_Box_Aus.Q OR rt_Box_Dauer.Q OR rt_Box_Intervall.Q OR rt_Box_Nachtr.Q OR rt_Box_Stocktemp.Q THEN
		xZielAus[2]       := HMI_OUT_Box_Aktuell_Aus;
		xZielDauer[2]     := HMI_OUT_Box_Aktuell_DauerbetriebEin;
		xZielIntervall[2] := HMI_OUT_Box_Aktuell_IntervallbetriebEIn;
		xZielNachtr[2]    := HMI_OUT_Box_Aktuell_NachtrocknungEin;
		xZielStocktemp[2] := HMI_OUT_Box_Aktuell_StocktemperaturEin;
		xUmschTrig[2]     := TRUE;
	END_IF;
	
	HMI_IN_Box_Aktuell_RestzeitUmschVerzBetriebsart := TO_UINT(gBetriebsparameter.Verzoegerungen.UmschaltungBetriebsartBox - TOF_Umsch[2].ET);
	//Aktuelle Trockengutfeuchte - Einstellung aus HMI
	gBetriebsparameter.Boxen[2].AktuelleTrockengutFeuchte := HMI_OUT_Box_Aktuell_TrockengutfeuchteAktuell;
	gBetriebsparameter.Boxen[2].StocktemperaturSoll := 	HMI_OUT_Box_Aktuell_StocktemperaturSoll;
		
	//PLC -> HMI
	HMI_IN_Box_Aktuell_Name := gBetriebsparameter.Boxen[2].NameBox;
	HMI_IN_Box_Aktuell_Temp := gStatusAnlage.AbluftBox2Temp;
	HMI_IN_Box_Aktuell_Feucht := gStatusAnlage.AbluftBox2Feuchte;	
	HMI_IN_Box_Aktuell_TrockengutIcon := gStatusAnlage.Box[2].TrockengutIcon;
	HMI_IN_Box_Aktuell_LaufRestzeitMinuten := gStatusAnlage.Box[2].LaufRestzeitMinuten;
	HMI_IN_Box_Aktuell_LaufRestzeitStunden := gStatusAnlage.Box[2].LaufRestzeitStunden;
	HMI_IN_Box_Aktuell_IconWitterung := gStatusAnlage.Box[2].IconWitterung;
	HMI_IN_Box_Aktuell_Status := TO_INT(gStatusAnlage.Box[2].Status);
	HMI_IN_Box_Aktuell_TextIndexLaufzeit := gStatusAnlage.Box[2].TextIndexLaufzeit;
	HMI_IN_Box_Aktuell_AnzeigeLaufRestzeit := gStatusAnlage.Box[2].AnzeigeLaufRestzeit;
	
ELSE 
	//nichts zu tun
END_IF;

IF (NOT gBetriebsparameter.Ausstattung.Box2) THEN
//--- Nur eine Box verfuegbar - Box 1 ist einzige Box : Betriebsartenwahl (flankengesteuert) ---
	firstStep := FALSE;
	rt_Box_Aus(CLK := HMI_OUT_Box1_Aus);
	rt_Box_Dauer(CLK := HMI_OUT_Box1_DauerbetriebEin);
	rt_Box_Intervall(CLK := HMI_OUT_Box1_IntervallbetriebEIn);
	rt_Box_Nachtr(CLK := HMI_OUT_Box1_NachtrocknungEin);
	rt_Box_Stocktemp(CLK := HMI_OUT_Box1_StocktemperaturEin);
	
	IF rt_Box_Aus.Q THEN
	    HMI_OUT_Box1_DauerbetriebEin     := FALSE;
	    HMI_OUT_Box1_IntervallbetriebEIn := FALSE;
	    HMI_OUT_Box1_NachtrocknungEin    := FALSE;
	    HMI_OUT_Box1_StocktemperaturEin  := FALSE;
	ELSIF rt_Box_Dauer.Q THEN
	    HMI_OUT_Box1_Aus                 := FALSE;
	    HMI_OUT_Box1_IntervallbetriebEIn := FALSE;
	    HMI_OUT_Box1_NachtrocknungEin    := FALSE;
	    HMI_OUT_Box1_StocktemperaturEin  := FALSE;
	ELSIF rt_Box_Intervall.Q THEN
	    HMI_OUT_Box1_Aus                 := FALSE;
	    HMI_OUT_Box1_DauerbetriebEin     := FALSE;
	    HMI_OUT_Box1_NachtrocknungEin    := FALSE;
	    HMI_OUT_Box1_StocktemperaturEin  := FALSE;
	ELSIF rt_Box_Nachtr.Q THEN
	    HMI_OUT_Box1_Aus                 := FALSE;
	    HMI_OUT_Box1_DauerbetriebEin     := FALSE;
	    HMI_OUT_Box1_IntervallbetriebEIn := FALSE;
	    HMI_OUT_Box1_StocktemperaturEin  := FALSE;
	ELSIF rt_Box_Stocktemp.Q THEN
	    HMI_OUT_Box1_Aus                 := FALSE;
	    HMI_OUT_Box1_DauerbetriebEin     := FALSE;
	    HMI_OUT_Box1_IntervallbetriebEIn := FALSE;
	    HMI_OUT_Box1_NachtrocknungEin 	 := FALSE;		
	END_IF;
	
	//--- Betriebsart verzögert übernehmen ---
	//--- Gewaehlte Betriebsart als Ziel merken + Hintergrund-Timer starten ---
	IF rt_Box_Aus.Q OR rt_Box_Dauer.Q OR rt_Box_Intervall.Q OR rt_Box_Nachtr.Q OR rt_Box_Stocktemp.Q THEN
		xZielAus[1]       := HMI_OUT_Box1_Aus;
		xZielDauer[1]     := HMI_OUT_Box1_DauerbetriebEin;
		xZielIntervall[1] := HMI_OUT_Box1_IntervallbetriebEIn;
		xZielNachtr[1]    := HMI_OUT_Box1_NachtrocknungEin;
		xZielStocktemp[1] := HMI_OUT_Box1_StocktemperaturEin;
		xUmschTrig[1]     := TRUE;
	END_IF;
	
	HMI_IN_Box1_RestzeitUmschVerzBetriebsart := TO_UINT(gBetriebsparameter.Verzoegerungen.UmschaltungBetriebsartBox - TOF_Umsch[1].ET);	
	
	//Aktuelle Trockengutfeuchte - Einstellung aus HMI
	gBetriebsparameter.Boxen[1].AktuelleTrockengutFeuchte := HMI_OUT_Box_Aktuell_TrockengutfeuchteAktuell;
	gBetriebsparameter.Boxen[1].StocktemperaturSoll := 	HMI_OUT_Box_Aktuell_StocktemperaturSoll;
	//Detailansicht Box 2
	
	//BOX 2 HIER EINFACH NUR GEH LOSSN!!! Wird in der VISU verwaltet!
	
END_IF;

//======================================================================
// Verzoegerte Betriebsart-Umschaltung (Hintergrund, eigener Timer je Box)
// - laeuft immer, auch wenn das Popup geschlossen ist
// - solange Timer laeuft bleibt die ALTE Betriebsart aktiv
// - erst nach Ablauf wird die neue Betriebsart uebernommen
//======================================================================
IF xInitUmsch THEN
	// Ziel = aktuell aktive Betriebsart -> kein Umschalten beim Anlauf
	FOR uIdx := 1 TO 2 DO
		xZielAus[uIdx]       := gBetriebsparameter.Boxen[uIdx].Aus;
		xZielDauer[uIdx]     := gBetriebsparameter.Boxen[uIdx].DauerbetriebEin;
		xZielIntervall[uIdx] := gBetriebsparameter.Boxen[uIdx].IntervallbetriebEin;
		xZielNachtr[uIdx]    := gBetriebsparameter.Boxen[uIdx].NachtrocknungEin;
		xZielStocktemp[uIdx] := gBetriebsparameter.Boxen[uIdx].StocktemperaturEin;
	END_FOR;
	xInitUmsch := FALSE;
END_IF;

FOR uIdx := 1 TO 2 DO
	TOF_Umsch[uIdx](IN := xUmschTrig[uIdx],
	                PT := gBetriebsparameter.Verzoegerungen.UmschaltungBetriebsartBox);
	xUmschTrig[uIdx] := FALSE;   // Trigger ist nur ein Puls (Timer haelt selbst nach)

	// Solange Timer laeuft (Q=TRUE) NICHT uebernehmen -> alte Betriebsart bleibt.
	// Nach Ablauf (Q=FALSE) neue Betriebsart uebernehmen.
	IF NOT TOF_Umsch[uIdx].Q THEN
		gBetriebsparameter.Boxen[uIdx].Aus                 := xZielAus[uIdx];
		gBetriebsparameter.Boxen[uIdx].DauerbetriebEin     := xZielDauer[uIdx];
		gBetriebsparameter.Boxen[uIdx].IntervallbetriebEin := xZielIntervall[uIdx];
		gBetriebsparameter.Boxen[uIdx].NachtrocknungEin    := xZielNachtr[uIdx];
		gBetriebsparameter.Boxen[uIdx].StocktemperaturEin  := xZielStocktemp[uIdx];
	END_IF;
END_FOR;

(*
-------------------------------------------------------------------------------
 SICHTBARKEITEN UND STATUS
-------------------------------------------------------------------------------
*)

//Lauf Restzeit einfach immer anzeigen
HMI_IN_Box1_AnzeigeLaufRestzeit := ICON_VISIBLE;
HMI_IN_Box2_AnzeigeLaufRestzeit := ICON_VISIBLE;

//Ventilator
IF gAlarmBetriebVentilator THEN 
	HMI_Ventilator1_FarbeIcon := ICON_ROT;
ELSIF gAktoren.xFrgVentilator THEN
	HMI_Ventilator1_FarbeIcon := ICON_GELB;
ELSE 
	HMI_Ventilator1_FarbeIcon := ICON_GRAU;
END_IF;

//Luftaufbereitung Icon
IF gBetriebsparameter.Ausstattung.Luftaufbereiter THEN 
	IF gAlarmBetriebLuftaufber THEN 
		Par_Luftaufbereitung_FarbeIcon := ICON_ROT;
	ELSIF gAktoren.xFrgLuftaufbereiter THEN
		Par_Luftaufbereitung_FarbeIcon := ICON_GELB;
	ELSE 
		Par_Luftaufbereitung_FarbeIcon := ICON_GRAU;
	END_IF;
ELSE 
	Par_Luftaufbereitung_FarbeIcon := ICON_HIDDEN;	
END_IF;

//Statusindex Textbox Luftaufbereiter PopUp
HMI_IN_LuftaufberStatusIndex := TO_USINT(gStatusAnlage.Aktor[AKTOR_LUFTAUFBER]);

//Abluftventilator
IF gBetriebsparameter.Ausstattung.Abluftventilator THEN 
	IF FALSE THEN //Abluftventilator hat keinen Alarm
		HMI_Abluft_FarbeIcon := ICON_ROT;
	ELSIF gAktoren.xFrgAbluftventilator THEN
		HMI_Abluft_FarbeIcon := ICON_GELB;
	ELSE 
		HMI_Abluft_FarbeIcon := ICON_GRAU;
	END_IF;
ELSE 
	HMI_Abluft_FarbeIcon := ICON_HIDDEN;	
END_IF;

// ===================== BOX 1 Status (Text fuer VISU) =====================
IF gCmdAnlage.Test THEN
    gStatusAnlage.Box[1].Status := STATUS_TESTBETRIEB;
ELSIF gBetriebsparameter.Boxen[1].Aus THEN
    gStatusAnlage.Box[1].Status := STATUS_STILLSTAND;
ELSIF gBetriebsparameter.Boxen[1].DauerbetriebEin THEN
    IF gStatusAnlage.Box[1].WetterIstSchlecht
       AND NOT (gBetriebsparameter.Ausstattung.Luftaufbereiter
                AND (gBetriebsparameter.Luftaufbereitung.Typ = HEIZREGISTER OR gBetriebsparameter.Luftaufbereitung.Typ = OFEN)
                AND (gBetriebsparameter.Luftaufbereitung.AutomatikbetriebEin OR gBetriebsparameter.Luftaufbereitung.DauerbetriebEin)) THEN
        IF gBetriebsparameter.Boxen[1].xBoxAktiv THEN
            gStatusAnlage.Box[1].Status := STATUS_SCHLECHTWETTER_LAUF;
        ELSE
            gStatusAnlage.Box[1].Status := STATUS_SCHLECHTWETTER_PAUSE;
        END_IF;
    ELSIF gBetriebsparameter.Boxen[1].xBoxAktiv THEN
        gStatusAnlage.Box[1].Status := STATUS_DAUERBETRIEB;
    ELSE
        gStatusAnlage.Box[1].Status := STATUS_DAUERBETRIEB_PAUSIERT;
    END_IF;
ELSIF gBetriebsparameter.Boxen[1].IntervallbetriebEin THEN
    IF gBetriebsparameter.Boxen[1].xBoxAktiv THEN
        gStatusAnlage.Box[1].Status := STATUS_INTERVALL_LAUF;
    ELSE
        gStatusAnlage.Box[1].Status := STATUS_INTERVALL_PAUSE;
    END_IF;
ELSIF gBetriebsparameter.Boxen[1].NachtrocknungEin THEN
    IF gBetriebsparameter.Boxen[1].xBoxAktiv THEN
        gStatusAnlage.Box[1].Status := STATUS_NACHTROCKNUNG_LAUF;
    ELSE
        gStatusAnlage.Box[1].Status := STATUS_NACHTROCKNUNG_PAUSE;
    END_IF;
ELSIF gBetriebsparameter.Boxen[1].StocktemperaturEin THEN
    IF gBetriebsparameter.Boxen[1].xBoxAktiv THEN
        gStatusAnlage.Box[1].Status := STATUS_STOCKTEMPERATUR_LAUF;       
    ELSE
        gStatusAnlage.Box[1].Status := STATUS_STOCKTEMPERATUR_PAUSE;
    END_IF;
ELSE
    gStatusAnlage.Box[1].Status := STATUS_STILLSTAND;
END_IF;

//BOX 2
// ===================== BOX 2 Status (Text fuer VISU) =====================
IF NOT gBetriebsparameter.Ausstattung.Box2 THEN
    gStatusAnlage.Box[2].Status := STATUS_NICHT_VERFUEGBAR;
ELSIF gCmdAnlage.Test THEN
    gStatusAnlage.Box[2].Status := STATUS_TESTBETRIEB;
ELSIF gBetriebsparameter.Boxen[2].Aus THEN
    gStatusAnlage.Box[2].Status := STATUS_STILLSTAND;
ELSIF gBetriebsparameter.Boxen[2].DauerbetriebEin THEN
    IF gStatusAnlage.Box[2].WetterIstSchlecht
       AND NOT (gBetriebsparameter.Ausstattung.Luftaufbereiter
                AND (gBetriebsparameter.Luftaufbereitung.Typ = HEIZREGISTER OR gBetriebsparameter.Luftaufbereitung.Typ = OFEN)
                AND (gBetriebsparameter.Luftaufbereitung.AutomatikbetriebEin OR gBetriebsparameter.Luftaufbereitung.DauerbetriebEin)) THEN
        IF gBetriebsparameter.Boxen[2].xBoxAktiv THEN
            gStatusAnlage.Box[2].Status := STATUS_SCHLECHTWETTER_LAUF;
        ELSE
            gStatusAnlage.Box[2].Status := STATUS_SCHLECHTWETTER_PAUSE;
        END_IF;
    ELSIF gBetriebsparameter.Boxen[2].xBoxAktiv THEN
        gStatusAnlage.Box[2].Status := STATUS_DAUERBETRIEB;
    ELSE
        gStatusAnlage.Box[2].Status := STATUS_DAUERBETRIEB_PAUSIERT;
    END_IF;
ELSIF gBetriebsparameter.Boxen[2].IntervallbetriebEin THEN
    IF gBetriebsparameter.Boxen[2].xBoxAktiv THEN
        gStatusAnlage.Box[2].Status := STATUS_INTERVALL_LAUF;
    ELSE
        gStatusAnlage.Box[2].Status := STATUS_INTERVALL_PAUSE;
    END_IF;
ELSIF gBetriebsparameter.Boxen[2].NachtrocknungEin THEN
    IF gBetriebsparameter.Boxen[2].xBoxAktiv THEN
        gStatusAnlage.Box[2].Status := STATUS_NACHTROCKNUNG_LAUF;
    ELSE
        gStatusAnlage.Box[2].Status := STATUS_NACHTROCKNUNG_PAUSE;
    END_IF;
ELSIF gBetriebsparameter.Boxen[2].StocktemperaturEin THEN
    IF gBetriebsparameter.Boxen[2].xBoxAktiv THEN
        gStatusAnlage.Box[2].Status := STATUS_STOCKTEMPERATUR_LAUF;
    ELSE
        gStatusAnlage.Box[2].Status := STATUS_STOCKTEMPERATUR_PAUSE;
    END_IF;
ELSE
    gStatusAnlage.Box[2].Status := STATUS_STILLSTAND;
END_IF;

(*
-------------------------------------------------------------------------------
 ALARME fuer Visu aufbereiten ARRAY -> UDINT Maske da Arrays nicht direkt
 an HMI gesendet werden koennen! 
-------------------------------------------------------------------------------
*)

//Reset Bitmasken vor Auswertung
HMI_IN_ALARM_WARNMASKE_1 := fcResetBitmask();
HMI_IN_ALARM_WARNMASKE_2 := fcResetBitmask();
HMI_IN_ALARM_STOERMASKE_1 := fcResetBitmask();
HMI_IN_ALARM_STOERMASKE_2 := fcResetBitmask();

//Array auf Bitmaske fuer HMI schreiben
FOR uIdx := 0 TO 31 DO
	//Erste Warnungsbitmaske [0.31]
	IF (gStatusAnlage.Alarm.ArrWarnung[uIdx]) THEN
		HMI_IN_ALARM_WARNMASKE_1:= fcSetBitInBitmask(Bitmask := HMI_IN_ALARM_WARNMASKE_1, BitNr:= uIdx);
	END_IF;
	//Zweite Warnungsbitmaske [32.63]
	IF (gStatusAnlage.Alarm.ArrWarnung[uIdx + 32]) THEN
		HMI_IN_ALARM_WARNMASKE_2:= fcSetBitInBitmask(Bitmask := HMI_IN_ALARM_WARNMASKE_2, BitNr:= uIdx);
	END_IF;	
	//Erste Stoerungsbitmaske [0.31]
	IF (gStatusAnlage.Alarm.ArrFehler[uIdx]) THEN
		HMI_IN_ALARM_STOERMASKE_1:= fcSetBitInBitmask(Bitmask := HMI_IN_ALARM_STOERMASKE_1, BitNr:= uIdx);
	END_IF;
	//Zweite Stoerungsbitmaske [32.63]
	IF (gStatusAnlage.Alarm.ArrFehler[uIdx + 32]) THEN
		HMI_IN_ALARM_STOERMASKE_2 := fcSetBitInBitmask(Bitmask := HMI_IN_ALARM_STOERMASKE_2, BitNr:= uIdx);
	END_IF;
END_FOR;
END_PROGRAM

PROGRAM StartStoppCyclic
  VAR
    xMindEineBoxAktiv : BOOL;
    xExternStart : BOOL;
    xExternStop : BOOL;
    xDauerbetriebBox1Anwahl : BOOL;
    xDauerbetriebBox2Anwahl : BOOL;
    xIntervallBox1Anwahl : BOOL;
    xIntervallBox2Anwahl : BOOL;
    xNachtrocknungBox1Anwahl : BOOL;
    xNachtrocknungBox2Anwahl : BOOL;
    xStocktemperaturBox1Anwahl : BOOL;
    xStocktemperaturBox2Anwahl : BOOL;
    xStocktemperaturBox1Aktiv : BOOL;
    xStocktemperaturBox2Aktiv : BOOL;
    xBox1Freigegeben : BOOL;
    xBox2Freigegeben : BOOL;
    xTarifStopWirksam : BOOL;
    usAktStunde : USINT;
    udIntervallMaskeBox1 : UDINT;
    udIntervallMaskeBox2 : UDINT;
    udNachtrocknungMaskeBox1 : UDINT;
    udNachtrocknungMaskeBox2 : UDINT;
    fbPulsPauseBox1 : fbPulsPause;
    xDauerbetriebBox1Trocknet : BOOL;
    xSchlechtwetterBox1Aktiv : BOOL;
    fbPulsPauseBox2 : fbPulsPause;
    xDauerbetriebBox2Trocknet : BOOL;
    xSchlechtwetterBox2Aktiv : BOOL;
    xStockHaltBox1 : BOOL := FALSE;  (* Haltebit Zweipunkt Box 1 *)
    xStockHaltBox2 : BOOL := FALSE;  (* Haltebit Zweipunkt Box 2 *)
    xLuftaufbAktiv : BOOL;  (* Heizregister oder Ofen vorhanden -> kein Puls/Pause *)
    xAnlageBetrieb : BOOL;
  END_VAR

(*
================================================================================
File        : StartStoppCyclic.st
Project     : CControl_Lite
Description :
    Start-/Stopp-Auswertung fuer 2-Box-Anlage.
    Ablauf: 
    	1) Betriebsarten  
    	2) Verriegelung  
    	3) Puls-/Pausebetrieb
        4) Boxaktivitaet  
        5) Start/Stopp
    Hinweis: BerechnungCyclic muss vor diesem Programm aufgerufen werden.
================================================================================
*)

(* ALLGEMEIN *)
usAktStunde := sysClock.hours;
udIntervallMaskeBox1 := Par_Box1_Intervallzeit;
udIntervallMaskeBox2 := Par_Box2_Intervallzeit;
udNachtrocknungMaskeBox1 := Par_Box1_Nachtrocknungszeit;
udNachtrocknungMaskeBox2 := Par_Box2_Nachtrocknungszeit;

xIntervallBox1Anwahl     := FALSE;
xIntervallBox2Anwahl     := FALSE;
xNachtrocknungBox1Anwahl := FALSE;
xNachtrocknungBox2Anwahl := FALSE;
xDauerbetriebBox1Anwahl  := FALSE;
xDauerbetriebBox2Anwahl  := FALSE;
xStocktemperaturBox1Anwahl  := FALSE;
xStocktemperaturBox2Anwahl  := FALSE;

(* Betriebsart *)
gCmdAnlage.Auto := NOT HMI_TEST_doIoTestAktivieren;
gCmdAnlage.Test := HMI_TEST_doIoTestAktivieren;


(*
================================================================================
 PHASE 1 - Betriebsarten ermitteln
 Prioritaet: Nachtrocknung > Intervallbetrieb > Dauerbetrieb
================================================================================
*)

//===== BOX 1 =====
IF gBetriebsparameter.Boxen[1].NachtrocknungEin AND (usAktStunde <= 23) THEN
	//Bitmaske um die aktuelle Stundenanzahl nach rechts schieben und pruefen ob Stunde in Maske aktiv
	xNachtrocknungBox1Anwahl := (SHR(IN := udNachtrocknungMaskeBox1, N := usAktStunde) AND 1) <> 0;
	
ELSIF gBetriebsparameter.Boxen[1].IntervallbetriebEin AND (usAktStunde <= 23) THEN
	xIntervallBox1Anwahl := (SHR(IN := udIntervallMaskeBox1, N := usAktStunde) AND 1) <> 0;
	
ELSIF gBetriebsparameter.Boxen[1].StocktemperaturEin THEN
	xStocktemperaturBox1Anwahl := TRUE;
	
ELSIF gBetriebsparameter.Boxen[1].DauerbetriebEin THEN
	xDauerbetriebBox1Anwahl := TRUE;
	
END_IF;

//===== BOX 2 =====
IF gBetriebsparameter.Boxen[2].NachtrocknungEin AND (usAktStunde <= 23) THEN
	xNachtrocknungBox2Anwahl := (SHR(IN := udNachtrocknungMaskeBox2, N := usAktStunde) AND 1) <> 0;

ELSIF gBetriebsparameter.Boxen[2].IntervallbetriebEin AND (usAktStunde <= 23) THEN
	xIntervallBox2Anwahl := (SHR(IN := udIntervallMaskeBox2, N := usAktStunde) AND 1) <> 0;

ELSIF gBetriebsparameter.Boxen[2].StocktemperaturEin THEN
	xStocktemperaturBox2Anwahl := TRUE;
	
ELSIF gBetriebsparameter.Boxen[2].DauerbetriebEin THEN
	xDauerbetriebBox2Anwahl := TRUE;
	
END_IF;


(*
================================================================================
 PHASE 2 - Verriegelung und Grundfreigabe
 Muss vor der Puls-/Pausezeit stehen, damit die Trocknungszeit nicht
 waehrend einer Sperre oder Stoerung abgezaehlt wird.
================================================================================
*)
                    
// Nachtrocknung hat Vorrang und uebersteuert die jeweils andere (aktive) Box.
// Bei beidseitiger Nachtrocknung mit ueberlappenden Stundenmasken laeuft nur Box 1.
xBox1Freigegeben := gCmdAnlage.Auto
                    AND NOT gCmdAnlage.FehlerStopp
                    AND NOT (xNachtrocknungBox2Anwahl AND NOT xNachtrocknungBox1Anwahl);

xBox2Freigegeben := gCmdAnlage.Auto
                    AND NOT gCmdAnlage.FehlerStopp
                    AND gBetriebsparameter.Ausstattung.Box2
                    AND NOT xNachtrocknungBox1Anwahl;

(*
================================================================================
 PHASE 3 - Stocktemperatur
 
================================================================================
*)
//===== BOX 1 - Stocktemperatur =====
IF xStocktemperaturBox1Anwahl THEN
    IF gStatusAnlage.StockTemperatur > (gBetriebsparameter.Boxen[1].StocktemperaturSoll + gBetriebsparameter.Boxen[1].StocktemperaturHysterese) THEN
    	xStockHaltBox1 := TRUE;
    ELSIF gStatusAnlage.StockTemperatur < (gBetriebsparameter.Boxen[1].StocktemperaturSoll - gBetriebsparameter.Boxen[1].StocktemperaturHysterese) THEN
        xStockHaltBox1 := FALSE;
    END_IF;
    xStocktemperaturBox1Aktiv := xStockHaltBox1;
ELSE
    xStockHaltBox1      := FALSE;
    xStocktemperaturBox1Aktiv := FALSE;
END_IF;
//===== BOX 2 - Stocktemperatur =====
IF xStocktemperaturBox2Anwahl THEN
    IF gStatusAnlage.StockTemperatur > (gBetriebsparameter.Boxen[2].StocktemperaturSoll + gBetriebsparameter.Boxen[2].StocktemperaturHysterese) THEN
        xStockHaltBox2 := TRUE;
    ELSIF gStatusAnlage.StockTemperatur < (gBetriebsparameter.Boxen[2].StocktemperaturSoll - gBetriebsparameter.Boxen[2].StocktemperaturHysterese) THEN
        xStockHaltBox2 := FALSE;
    END_IF;
    xStocktemperaturBox2Aktiv := xStockHaltBox2;
ELSE
    xStockHaltBox2      := FALSE;
    xStocktemperaturBox2Aktiv := FALSE;
END_IF;


(*
================================================================================
 PHASE 4 - Schlechtwetter Puls-/Pausebetrieb
 Wirkt ausschliesslich auf den Dauerbetrieb. Intervall- und Nachtrocknungs-
 betrieb laufen unveraendert nach Stundenmaske.
================================================================================
*)

//Luftaufbereitung aktiv (Heizregister oder Ofen laeuft in Automatik- oder
//Dauerbetrieb) -> im Automatikbetrieb durchgehend trocknen statt Lauf/Pause.
//Ausnahme: Stellt der Bediener die Luftaufbereitung auf AUS (weder Automatik-
//noch Dauerbetrieb), soll die Witterung mit dem Lauf/Pause-Programm wieder
//greifen -> dann gilt die Luftaufbereitung als nicht aktiv.
//Bewusst ueber die aktiven Betriebsarten abgefragt (nicht ueber '.Aus'), da beim
//Steuerungsstart nicht sicher ist, dass '.Aus' gesetzt ist.
xLuftaufbAktiv := gBetriebsparameter.Ausstattung.Luftaufbereiter
                  AND (gBetriebsparameter.Luftaufbereitung.Typ = HEIZREGISTER
                       OR gBetriebsparameter.Luftaufbereitung.Typ = OFEN)
                  AND (gBetriebsparameter.Luftaufbereitung.AutomatikbetriebEin
                       OR gBetriebsparameter.Luftaufbereitung.DauerbetriebEin);

//===== BOX 1 =====
xSchlechtwetterBox1Aktiv := xDauerbetriebBox1Anwahl
                            AND xBox1Freigegeben
                            AND gStatusAnlage.Box[1].WetterIstSchlecht
                            AND (gStatusAnlage.Box[1].AktSchlechtwetterPause <> 0)
                            AND NOT xLuftaufbAktiv;

fbPulsPauseBox1.Freigabe      := xSchlechtwetterBox1Aktiv;
fbPulsPauseBox1.StartMitPause := FALSE;   //bei Wetterumschlag zuerst trocknen
fbPulsPauseBox1.ZeitPuls      := gStatusAnlage.Box[1].AktSchlechtwetterPuls;
fbPulsPauseBox1.ZeitPause     := gStatusAnlage.Box[1].AktSchlechtwetterPause;
fbPulsPauseBox1();

gStatusAnlage.Box[1].SchlechtwetterPulsOut   := fbPulsPauseBox1.PulsOut;
gStatusAnlage.Box[1].SchlechtwetterPauseOut  := fbPulsPauseBox1.PauseOut;
gStatusAnlage.Box[1].RestSchlechtwetterPuls  := fbPulsPauseBox1.RestzeitPuls;
gStatusAnlage.Box[1].RestSchlechtwetterPause := fbPulsPauseBox1.RestzeitPause;

IF xSchlechtwetterBox1Aktiv THEN
	//Schlechtwetter: nur waehrend der Pulszeit trocknen
	xDauerbetriebBox1Trocknet := fbPulsPauseBox1.PulsOut;
ELSE
	//Schoenwetter oder keine Pausezeit parametriert: Dauerbetrieb
	xDauerbetriebBox1Trocknet := xDauerbetriebBox1Anwahl;
END_IF;

//===== BOX 2 =====
xSchlechtwetterBox2Aktiv := xDauerbetriebBox2Anwahl
                            AND xBox2Freigegeben
                            AND gStatusAnlage.Box[2].WetterIstSchlecht
                            AND (gStatusAnlage.Box[2].AktSchlechtwetterPause <> 0)
                            AND NOT xLuftaufbAktiv;

fbPulsPauseBox2.Freigabe      := xSchlechtwetterBox2Aktiv;
fbPulsPauseBox2.StartMitPause := FALSE;
fbPulsPauseBox2.ZeitPuls      := gStatusAnlage.Box[2].AktSchlechtwetterPuls;
fbPulsPauseBox2.ZeitPause     := gStatusAnlage.Box[2].AktSchlechtwetterPause;
fbPulsPauseBox2();

gStatusAnlage.Box[2].SchlechtwetterPulsOut   := fbPulsPauseBox2.PulsOut;
gStatusAnlage.Box[2].SchlechtwetterPauseOut  := fbPulsPauseBox2.PauseOut;
gStatusAnlage.Box[2].RestSchlechtwetterPuls  := fbPulsPauseBox2.RestzeitPuls;
gStatusAnlage.Box[2].RestSchlechtwetterPause := fbPulsPauseBox2.RestzeitPause;

IF xSchlechtwetterBox2Aktiv THEN
	xDauerbetriebBox2Trocknet := fbPulsPauseBox2.PulsOut;
ELSE
	xDauerbetriebBox2Trocknet := xDauerbetriebBox2Anwahl;
END_IF;


(*
================================================================================
 PHASE 5 - Boxaktivitaet
================================================================================
*)

gBetriebsparameter.Boxen[1].xBoxAktiv := (xDauerbetriebBox1Trocknet
                                          OR xIntervallBox1Anwahl
                                          OR xNachtrocknungBox1Anwahl
                                          OR xStocktemperaturBox1Aktiv)
                                         AND xBox1Freigegeben;

gBetriebsparameter.Boxen[2].xBoxAktiv := (xDauerbetriebBox2Trocknet
                                          OR xIntervallBox2Anwahl
                                          OR xNachtrocknungBox2Anwahl
                                          OR xStocktemperaturBox2Aktiv)
                                         AND xBox2Freigegeben;

xMindEineBoxAktiv := gBetriebsparameter.Boxen[1].xBoxAktiv
                     OR gBetriebsparameter.Boxen[2].xBoxAktiv;


(*
================================================================================
 PHASE 6 - Start/Stopp
================================================================================
*)

(* externe Signale optional, muessen beschrieben werden wenn gewuenscht *)
xExternStart := gCmdAnlage.StartExtern;
xExternStop  := gCmdAnlage.StoppExtern;

(* Fehlerstopp vorerst ohne Alarmmatrix, Variable wird in AlarmCyclic beschrieben *)
//gCmdAnlage.FehlerStopp := FALSE;

//Anlage laeuft solange eine Box aktiv ODER die Luftaufbereitung noch auskuehlt
xAnlageBetrieb := xMindEineBoxAktiv OR gAktoren.xLuftaufbNachlauf;

//Tarifabschaltung wirkt erst, wenn Luftaufbereitung/Auskuehlung/Betriebsmeldung
//abgeschlossen sind (diese haben Vorrang).
xTarifStopWirksam := gCmdAnlage.xTarifAbschaltung AND NOT gAktoren.xLuftaufbNachlauf;

gCmdAnlage.Start := gCmdAnlage.Auto
                    AND (xAnlageBetrieb OR xExternStart)
                    AND NOT gCmdAnlage.FehlerStopp
                    AND NOT xTarifStopWirksam;

gCmdAnlage.Stopp := gCmdAnlage.Auto
                    AND ((NOT xAnlageBetrieb) OR xExternStop
                         OR gCmdAnlage.FehlerStopp
                         OR xTarifStopWirksam);
END_PROGRAM

PROGRAM BackgroundTask
  VAR
    retVal : USINT;
  END_VAR

//SetSysClock (Anforderung kommt von HMI)
IF HMI_OUT_SysClock_ReqSet THEN 
  //Uhrzeit setzen
  retVal :=	sysClockWrite(
  						  seconds 	:= TO_USINT(HMI_OUT_SysClock_seconds), 
						  minutes 	:= TO_USINT(HMI_OUT_SysClock_minutes),
						  hours 	:= TO_USINT(HMI_OUT_SysClock_hours),
						  dayweek 	:= TO_USINT(HMI_OUT_SysClock_dayweek),
						  daymonth 	:= TO_USINT(HMI_OUT_SysClock_daymonth), 
						  month 	:= TO_USINT(HMI_OUT_SysClock_month), 
						  year 		:= TO_USINT(HMI_OUT_SysClock_year)
						  );
	
END_IF;

IF retVal <> 0 THEN
	HMI_OUT_SysClock_ReqSet := FALSE;
	retVal := 0;
END_IF;
END_PROGRAM

FUNCTION_BLOCK fbBoxenklappe
  VAR
    uiStep : UINT := 0;
    stateEntry : BOOL := TRUE;
    TON_Laufzeit : TON;
    TON_AnzVerz : TON;
  END_VAR
  VAR_INPUT
    Oeffnen : BOOL;
    Schliessen : BOOL;
    EndlageOffen : BOOL;
    EndlageGeschl : BOOL;
    EndlagenVhd : BOOL;
    LaufzeitOeffnen : UDINT;
    LaufzeitSchliessen : UDINT;
    Stoerung : BOOL;
    QuitFehler : BOOL;
  END_VAR
  VAR_OUTPUT
    OeffnenOut : BOOL;
    SchliessenOut : BOOL;
    KlappeIstOffenOut : BOOL;
    KlappeIstGeschlOut : BOOL;
    FehlerLaufzeitOeffnen : BOOL;
    FehlerLaufzeitSchliessen : BOOL;
  END_VAR

(*
================================================================================
 File        : fbBoxenklappe.st
 Project     : CControl_Lite
 Controller  : Schneider / EcoStruxure Machine Expert HVAC
 Author      : RIG Automation
 Created     : 2026-04-03
 Version     : V0.02
 Description :
    Funktionsbaustein zur Ansteuerung einer Boxenklappe mit einem Wechsler-
    Relais.

    Funktionsprinzip:
      - nicht angesteuert = Richtung A
      - angesteuert       = Richtung B

    Für die Anwendung in CControl_Lite gilt:
      - OeffnenOut     = TRUE
      - SchliessenOut  = FALSE

    Funktionsumfang:
      - Laufzeitüberwachung Öffnen/Schließen
      - Fehlerquittierung
      - Endlagenbehandlung
      - Betrieb auch ohne Endlagen möglich
      - 40 ms Anzugsverzögerung

================================================================================
 Change History
--------------------------------------------------------------------------------
 Version | Date       | Author          | Description
--------------------------------------------------------------------------------
 V0.02   | 2026-04-03 | RIG Automation  | Initialerstellung
================================================================================
*)

IF (NOT Stoerung) THEN

    (*
    ---------------------------------------------------------------------------
    Fehlerquittierung Laufzeitüberwachung
    ---------------------------------------------------------------------------
    *)
    IF QuitFehler OR (LaufzeitOeffnen = 0) OR (NOT EndlagenVhd) THEN
        FehlerLaufzeitOeffnen := FALSE;
    END_IF;

    IF QuitFehler OR (LaufzeitSchliessen = 0) OR (NOT EndlagenVhd) THEN
        FehlerLaufzeitSchliessen := FALSE;
    END_IF;


    CASE uiStep OF

        (*
        =======================================================================
        WARTEN
        =======================================================================
        *)
        0:
            (* state entry *)
            IF stateEntry THEN
                stateEntry := FALSE;
                TON_Laufzeit(IN := FALSE, PT := 0);
                TON_AnzVerz(IN := FALSE, PT := 0);
            END_IF;

            (* state during *)
            IF QuitFehler OR (LaufzeitOeffnen = 0) OR (NOT EndlagenVhd) THEN
                FehlerLaufzeitOeffnen := FALSE;
            END_IF;

            IF QuitFehler OR (LaufzeitSchliessen = 0) OR (NOT EndlagenVhd) THEN
                FehlerLaufzeitSchliessen := FALSE;
            END_IF;

            (* state exit *)
            (*
            IF EndlagenVhd OR (LaufzeitOeffnen = 0) THEN
                IF Oeffnen AND NOT FehlerLaufzeitOeffnen THEN
                    stateEntry := TRUE;
                    uiStep  := 1;
                END_IF;
            ELSE
                IF Oeffnen AND NOT KlappeIstOffenOut THEN
                    stateEntry := TRUE;
                    uiStep  := 1;
                END_IF;
            END_IF;

            IF EndlagenVhd OR (LaufzeitSchliessen = 0) THEN
                IF Schliessen AND NOT FehlerLaufzeitSchliessen THEN
                    stateEntry := TRUE;
                    uiStep  := 2;
                END_IF;
            ELSE
                IF Schliessen AND NOT KlappeIstGeschlOut THEN
                    stateEntry := TRUE;
                    uiStep := 2;
                END_IF;
            END_IF;
            *)
            
            (* state exit *)
			IF EndlagenVhd THEN
			    IF Oeffnen AND NOT FehlerLaufzeitOeffnen THEN
			        stateEntry := TRUE;
			        uiStep  := 1;
			    END_IF;
			ELSE
			    IF Oeffnen AND NOT KlappeIstOffenOut THEN     // ohne Endlagen IMMER zeitbasiert (auch Laufzeit=0)
			        stateEntry := TRUE;
			        uiStep  := 1;
			    END_IF;
			END_IF;
			
			IF EndlagenVhd THEN
			    IF Schliessen AND NOT FehlerLaufzeitSchliessen THEN
			        stateEntry := TRUE;
			        uiStep  := 2;
			    END_IF;
			ELSE
			    IF Schliessen AND NOT KlappeIstGeschlOut THEN
			        stateEntry := TRUE;
			        uiStep := 2;
			    END_IF;
			END_IF;


        (*
        =======================================================================
        OEFFNEN
        =======================================================================
        *)
        1:
            (* state entry *)
            IF stateEntry THEN
                stateEntry := FALSE;
                TON_Laufzeit(IN := FALSE, PT := 0);
                TON_AnzVerz(IN := FALSE, PT := 0);
                FehlerLaufzeitOeffnen := FALSE;
                FehlerLaufzeitSchliessen := FALSE;
                SchliessenOut := FALSE;
                KlappeIstGeschlOut := FALSE;
                KlappeIstOffenOut := FALSE;
            END_IF;

            (* state during *)
            (*
            TON_Laufzeit(IN := OeffnenOut AND NOT EndlageOffen, PT := LaufzeitOeffnen);
            *)            
            TON_Laufzeit(IN := OeffnenOut AND (NOT EndlageOffen OR NOT EndlagenVhd), PT := LaufzeitOeffnen);
            TON_AnzVerz(IN := TRUE, PT := 40);
            OeffnenOut := TON_AnzVerz.Q;

            (* state exit *)
            (*
            IF (NOT Oeffnen) OR Schliessen OR (TON_Laufzeit.Q AND (LaufzeitOeffnen <> 0)) THEN
                IF (TON_Laufzeit.Q AND (LaufzeitOeffnen <> 0) AND NOT EndlagenVhd) THEN
                    KlappeIstOffenOut := TRUE;
                ELSIF (TON_Laufzeit.Q AND (LaufzeitOeffnen <> 0)) THEN
                    FehlerLaufzeitOeffnen := TRUE;
                END_IF;

                stateEntry := TRUE;
                uiStep  := 0;
            END_IF;
            *)
            
            (* state exit *)
			IF (NOT Oeffnen) OR Schliessen OR (TON_Laufzeit.Q AND (LaufzeitOeffnen <> 0))
			    OR (NOT EndlagenVhd AND (LaufzeitOeffnen = 0)) THEN
			    IF (NOT EndlagenVhd) AND (TON_Laufzeit.Q OR (LaufzeitOeffnen = 0)) THEN
			        KlappeIstOffenOut := TRUE;            // ohne Endlagen: nach Laufzeit ODER sofort (Laufzeit=0)
			    ELSIF (TON_Laufzeit.Q AND (LaufzeitOeffnen <> 0)) THEN
			        FehlerLaufzeitOeffnen := TRUE;        // mit Endlagen: Laufzeitueberschreitung = Fehler
			    END_IF;
			
			    stateEntry := TRUE;
			    uiStep  := 0;
			END_IF;


        (*
        =======================================================================
        SCHLIESSEN
        =======================================================================
        *)
        2:
            (* state entry *)
            IF stateEntry THEN
                stateEntry := FALSE;
                TON_Laufzeit(IN := FALSE, PT := 0);
                TON_AnzVerz(IN := FALSE, PT := 0);
                FehlerLaufzeitOeffnen := FALSE;
                FehlerLaufzeitSchliessen := FALSE;
                OeffnenOut := FALSE;
                KlappeIstGeschlOut := FALSE;
                KlappeIstOffenOut := FALSE;
            END_IF;

            (* state during *)
            //TON_Laufzeit(IN := SchliessenOut AND NOT EndlageGeschl, PT := LaufzeitSchliessen);
            TON_Laufzeit(IN := SchliessenOut AND (NOT EndlageGeschl OR NOT EndlagenVhd), PT := LaufzeitSchliessen);
            TON_AnzVerz(IN := TRUE, PT := 40);
            SchliessenOut := TON_AnzVerz.Q;

            (* state exit *)(*
            IF (NOT Schliessen) OR Oeffnen OR (TON_Laufzeit.Q AND (LaufzeitSchliessen <> 0)) THEN
                IF (TON_Laufzeit.Q AND (LaufzeitSchliessen <> 0) AND NOT EndlagenVhd) THEN
                    KlappeIstGeschlOut := TRUE;
                ELSIF (TON_Laufzeit.Q AND (LaufzeitSchliessen <> 0)) THEN
                    FehlerLaufzeitSchliessen := TRUE;
                END_IF;

                stateEntry := TRUE;
                uiStep := 0;
            END_IF;
            *)
            (* state exit *)
			IF (NOT Schliessen) OR Oeffnen OR (TON_Laufzeit.Q AND (LaufzeitSchliessen <> 0))
			    OR (NOT EndlagenVhd AND (LaufzeitSchliessen = 0)) THEN
			    IF (NOT EndlagenVhd) AND (TON_Laufzeit.Q OR (LaufzeitSchliessen = 0)) THEN
			        KlappeIstGeschlOut := TRUE;
			    ELSIF (TON_Laufzeit.Q AND (LaufzeitSchliessen <> 0)) THEN
			        FehlerLaufzeitSchliessen := TRUE;
			    END_IF;
			
			    stateEntry := TRUE;
			    uiStep := 0;
			END_IF;

    END_CASE;

ELSE
    OeffnenOut := FALSE;
    SchliessenOut := FALSE;
    stateEntry := TRUE;
    FehlerLaufzeitOeffnen := FALSE;
    FehlerLaufzeitSchliessen := FALSE;
    KlappeIstGeschlOut := FALSE;
    KlappeIstOffenOut := FALSE;
    uiStep := 0;
END_IF;
END_FUNCTION_BLOCK

FUNCTION_BLOCK fbTrockStrombegr
  VAR
    FreigZeitfenster1 : BOOL;
    FreigZeitfenster2 : BOOL;
    FreigZeitfenster3 : BOOL;
  END_VAR
  VAR_INPUT
    Freigabe : BOOL;  (* Freigabe Strombegrenzung *)
    StartZeit1 : REAL;  (* Startzeit Zeitfenster 1 *)
    StoppZeit1 : REAL;  (* Stoppzeit Zeitfenster 1 *)
    AktZeit : REAL;  (* aktuelle Uhrzeit *)
    StartZeit2 : REAL;
    StoppZeit2 : REAL;
    StartZeit3 : REAL;
    StoppZeit3 : REAL;
    DrehzahlBegrenzung1 : REAL;  (* Drehzahlbegrenzung Zeitfenster 1 *)
    DrehzahlBegrenzung2 : REAL;  (* Drehzahlbegrenzung Zeitfenster 2 *)
    DrehzahlBegrenzung3 : REAL;  (* Drehzahlbegrenzung Zeitfenster 3 *)
  END_VAR
  VAR_OUTPUT
    StrombegrenzungEin : BOOL;  (* Strombegrenzung aktiv *)
    DrehzahlBegrenzung : REAL;  (* wirksame Drehzahlbegrenzung *)
  END_VAR

IF (Freigabe = TRUE) THEN
    // Zeitfenster 1 ********************************************************
    FreigZeitfenster1 := FALSE;
    IF (StartZeit1 > StoppZeit1) THEN
        IF (AktZeit >= StartZeit1) OR (AktZeit < StoppZeit1) THEN
            FreigZeitfenster1 := TRUE;
        END_IF;
    ELSE
        IF (AktZeit >= StartZeit1) AND (AktZeit < StoppZeit1) THEN
            FreigZeitfenster1 := TRUE;
        END_IF;
    END_IF;
    // Zeitfenster 2 ********************************************************
    FreigZeitfenster2 := FALSE;
    IF (StartZeit2 > StoppZeit2) THEN
        IF (AktZeit >= StartZeit2) OR (AktZeit < StoppZeit2) THEN
            FreigZeitfenster2 := TRUE;
        END_IF;
    ELSE
        IF (AktZeit >= StartZeit2) AND (AktZeit < StoppZeit2) THEN
            FreigZeitfenster2 := TRUE;
        END_IF;
    END_IF;
    // Zeitfenster 3 ********************************************************
    FreigZeitfenster3 := FALSE;
    IF (StartZeit3 > StoppZeit3) THEN
        IF (AktZeit >= StartZeit3) OR (AktZeit < StoppZeit3) THEN
            FreigZeitfenster3 := TRUE;
        END_IF;
    ELSE
        IF (AktZeit >= StartZeit3) AND (AktZeit < StoppZeit3) THEN
            FreigZeitfenster3 := TRUE;
        END_IF;
    END_IF;
    // Drehzahlbegrenzungen 1 - 3
    IF (FreigZeitfenster1) THEN
        DrehzahlBegrenzung := DrehzahlBegrenzung1;
    ELSIF (FreigZeitfenster2) THEN
        DrehzahlBegrenzung := DrehzahlBegrenzung2;
    ELSIF (FreigZeitfenster3) THEN
        DrehzahlBegrenzung := DrehzahlBegrenzung3;
    ELSE
        DrehzahlBegrenzung := 0.0;
    END_IF;
    StrombegrenzungEin := FreigZeitfenster1 OR FreigZeitfenster2 OR FreigZeitfenster3;
ELSE
    FreigZeitfenster1  := FALSE;
    FreigZeitfenster2  := FALSE;
    FreigZeitfenster3  := FALSE;
    StrombegrenzungEin := FALSE;
    DrehzahlBegrenzung := 0.0;
END_IF;
END_FUNCTION_BLOCK

FUNCTION_BLOCK fbBoxenWLO
  VAR
    uStep : USINT;  (* Schrittkette 0..2 *)
    stateEntry : BOOL;  (* Entry-Flag Schritt *)
    TON_VerzBetriebsmeldung : TON;
    TOF_Auskuehlzeit : TOF;
    loc_WetterIstSchlecht : BOOL;
    loc_WetterIstGut : BOOL;
    TON_WetterIstGut : TON;
    TON_WetterIstSchlecht : TON;
    R_TRIG_WetterIstGut : R_TRIG;  (* ersetzt EDGEPOS *)
    R_TRIG_WetterIstSchlecht : R_TRIG;  (* ersetzt EDGEPOS *)
  END_VAR
  VAR_INPUT
    Freigabe : BOOL;  (* Grundfreigabe Baustein *)
    Automatikbetrieb : BOOL;  (* Betriebsart Automatik (witterungsgeführt) *)
    Dauerbetrieb : BOOL;  (* Betriebsart Dauerbetrieb *)
    FehlerSensorAussenluft : BOOL;  (* Eingang Sensorfehler Frischluft *)
    FrischluftSattDefizitIst : REAL;  (* Ist-Sättigungsdefizit *)
    FrischluftSattDefizitSoll : REAL;  (* Soll-Sättigungsdefizit *)
    Hysterese : REAL;  (* Hysterese Sättigungsdefizit *)
    UmschaltverzWitterung : UDINT;  (* Umschaltverzögerung gut/schlecht [ms] *)
    WarmlufttemperaturVorgabe : REAL;  (* Solltemperatur-Vorgabe (HMI) *)
    OptionBetriebsmldgVhd : BOOL;  (* Option Betriebsmeldung vorhanden *)
    BetriebsmeldungWarmluftofen : BOOL;  (* Rückmeldung Brenner/Ofen läuft *)
    VerzBetriebsmeldung : UDINT;  (* Zündzeit / Überwachungsverzögerung [ms] *)
    Auskuehlzeit : UDINT;  (* Nachlauf-/Auskühlzeit [ms] *)
    QuitFehler : BOOL;  (* Fehlerquittierung *)
    WetterIstSchlecht : BOOL;  (* externe Vorgabe Wetter schlecht *)
  END_VAR
  VAR_OUTPUT
    FreigabeWarmluftofenOut : BOOL;  (* Freigabe an Ofen *)
    WarmlufttempSollOut : REAL;  (* ausgegebene Solltemperatur *)
    FehlerBetriebsmeldungOut : BOOL;  (* gespeicherter Fehler Betriebsmeldung *)
    FehlerSensorAussenluftOut : BOOL;  (* gespeicherter Sensorfehler *)
    WarmluftofenAktiv : BOOL;  (* Ofen aktiv (inkl. Auskühlung) *)
    RestAuskuehlzeit : UDINT;  (* Restlaufzeit Auskühlung [ms] für Visu *)
  END_VAR

//Auskühlzeit Warmluftofen, wenn Option Betriebsmeldung nicht vorhanden
TOF_Auskuehlzeit(IN := FreigabeWarmluftofenOut, PT := Auskuehlzeit);

//Restlaufzeit Auskühlung berechnen (für Visu)
RestAuskuehlzeit := Auskuehlzeit - TO_UDINT(TOF_Auskuehlzeit.ET);

//Ausgang für Warmluftofen aktiv
WarmluftofenAktiv := (TOF_Auskuehlzeit.Q AND NOT OptionBetriebsmldgVhd)
                     OR (BetriebsmeldungWarmluftofen AND OptionBetriebsmldgVhd)
                     OR FreigabeWarmluftofenOut;

//Fehlerquittierung
IF QuitFehler THEN
    FehlerSensorAussenluftOut := FALSE;
    FehlerBetriebsmeldungOut  := FALSE;
END_IF;


IF Freigabe THEN

    CASE uStep OF

        //AUS *********************************************************************************************
        0:
            IF stateEntry THEN
                stateEntry              := FALSE;
                FreigabeWarmluftofenOut := FALSE;
                WarmlufttempSollOut     := 0.0;
                TON_VerzBetriebsmeldung(IN := FALSE, PT := 0);
            END_IF;

            //Automatikbetrieb aktiviert
            IF Automatikbetrieb AND NOT FehlerSensorAussenluftOut AND NOT FehlerBetriebsmeldungOut AND NOT FehlerSensorAussenluft THEN
                stateEntry := TRUE;
                uStep       := 1;
            ELSIF Dauerbetrieb AND NOT FehlerSensorAussenluftOut AND NOT FehlerBetriebsmeldungOut THEN
                stateEntry := TRUE;
                uStep       := 2;
            END_IF;


        //AUTOMATIKBETRIEB ********************************************************************************
        1:
            IF stateEntry THEN
                stateEntry := FALSE;
                TON_VerzBetriebsmeldung(IN := FALSE, PT := 0);
            END_IF;

            //Bei Neustart (Wetter nicht gut oder schlecht) ohne Verzögerung umschalten
            IF NOT loc_WetterIstSchlecht AND NOT loc_WetterIstGut THEN
                IF (FrischluftSattDefizitIst < FrischluftSattDefizitSoll) THEN
                    loc_WetterIstSchlecht := TRUE;
                ELSIF (FrischluftSattDefizitIst >= FrischluftSattDefizitSoll) THEN
                    loc_WetterIstGut := TRUE;
                END_IF;
            END_IF;

            //Umschaltverzögerung gutes Wetter / schlechtes Wetter
            TON_WetterIstGut(IN := loc_WetterIstSchlecht AND (FrischluftSattDefizitIst >= (FrischluftSattDefizitSoll + Hysterese)), PT := UmschaltverzWitterung);
            TON_WetterIstSchlecht(IN := loc_WetterIstGut AND (FrischluftSattDefizitIst < (FrischluftSattDefizitSoll - Hysterese)), PT := UmschaltverzWitterung);

            //Flankenauswertung (ersetzt EDGEPOS)
            R_TRIG_WetterIstGut(CLK := TON_WetterIstGut.Q);
            R_TRIG_WetterIstSchlecht(CLK := TON_WetterIstSchlecht.Q);

            IF R_TRIG_WetterIstGut.Q THEN
                loc_WetterIstGut      := TRUE;
                loc_WetterIstSchlecht := FALSE;
            ELSIF R_TRIG_WetterIstSchlecht.Q THEN
                loc_WetterIstGut      := FALSE;
                loc_WetterIstSchlecht := TRUE;
            END_IF;

            //Freigabe Warmluftofen
            FreigabeWarmluftofenOut := loc_WetterIstSchlecht OR WetterIstSchlecht;
            WarmlufttempSollOut     := WarmlufttemperaturVorgabe;

            //Verzögerung Überwachung Betriebsmeldung (Zündzeit)
            TON_VerzBetriebsmeldung(IN := FreigabeWarmluftofenOut AND OptionBetriebsmldgVhd
                              			  AND NOT BetriebsmeldungWarmluftofen
                            			  AND (VerzBetriebsmeldung > 0),
                        			PT := VerzBetriebsmeldung);

            //Fehler keine Betriebsmeldung
            IF TON_VerzBetriebsmeldung.Q THEN
                FehlerBetriebsmeldungOut := TRUE;
                stateEntry := TRUE;
                uStep       := 0;
            //Fehler Sensor Frischluft
            ELSIF FehlerSensorAussenluft THEN
                FehlerSensorAussenluftOut := TRUE;
                stateEntry := TRUE;
                uStep       := 0;
            //Dauerbetrieb aktiv
            ELSIF Dauerbetrieb THEN
                stateEntry := TRUE;
                uStep       := 2;
            //Kein Automatikbetrieb
            ELSIF NOT Automatikbetrieb THEN
                stateEntry := TRUE;
                uStep       := 0;
            END_IF;


        //DAUERBETRIEB ***********************************************************************************
        2:
            IF stateEntry THEN
                stateEntry := FALSE;
                TON_VerzBetriebsmeldung(IN := FALSE, PT := 0);
            END_IF;

            //Freigabe Warmluftofen
            FreigabeWarmluftofenOut := TRUE;
            WarmlufttempSollOut     := WarmlufttemperaturVorgabe;

            //Verzögerung Überwachung Betriebsmeldung (Zündzeit)
            TON_VerzBetriebsmeldung(IN := FreigabeWarmluftofenOut AND OptionBetriebsmldgVhd AND NOT BetriebsmeldungWarmluftofen, PT := VerzBetriebsmeldung);

            //Fehler
            IF TON_VerzBetriebsmeldung.Q THEN
                FehlerBetriebsmeldungOut := TRUE;
                stateEntry := TRUE;
                uStep       := 0;
            //Automatikbetrieb aktiv
            ELSIF Automatikbetrieb THEN
                stateEntry := TRUE;
                uStep       := 1;
            //Kein Dauerbetrieb
            ELSIF NOT Dauerbetrieb THEN
                stateEntry := TRUE;
                uStep       := 0;
            END_IF;

    END_CASE;

ELSE

    FreigabeWarmluftofenOut   := FALSE;
    WarmlufttempSollOut       := 0.0;
    uStep                      := 0;
    stateEntry                := TRUE;
    FehlerSensorAussenluftOut := FALSE;
    FehlerBetriebsmeldungOut  := FALSE;

END_IF;
END_FUNCTION_BLOCK

FUNCTION_BLOCK fbHeizregister
  VAR
    uStep : USINT;  (* Schrittkette 0..2 *)
    stateEntry : BOOL;  (* Entry-Flag Schritt *)
    loc_WetterIstSchlecht : BOOL;
    loc_WetterIstGut : BOOL;
    TON_WetterIstGut : TON;
    TON_WetterIstSchlecht : TON;
    R_TRIG_WetterIstGut : R_TRIG;  (* ersetzt EDGEPOS *)
    R_TRIG_WetterIstSchlecht : R_TRIG;  (* ersetzt EDGEPOS *)
  END_VAR
  VAR_INPUT
    Freigabe : BOOL;  (* Grundfreigabe Baustein *)
    QuitFehler : BOOL;  (* Fehlerquittierung *)
    Automatikbetrieb : BOOL;  (* Betriebsart Automatik (witterungsgeführt) *)
    Dauerbetrieb : BOOL;  (* Betriebsart Dauerbetrieb *)
    FehlerSensorAussenluft : BOOL;  (* Eingang Sensorfehler Frischluft *)
    FrischluftSattDefizitIst : REAL;  (* Ist-Sättigungsdefizit *)
    FrischluftSattDefizitSoll : REAL;  (* Soll-Sättigungsdefizit *)
    Hysterese : REAL;  (* Hysterese Sättigungsdefizit *)
    UmschaltverzWitterung : UDINT;  (* Umschaltverzögerung gut/schlecht [ms] *)
    WetterIstSchlecht : BOOL;  (* externe Vorgabe Wetter schlecht *)
    DrehzahlHeizregisterSoll : REAL;  (* Drehzahlvorgabe Heizungspumpe (Soll) *)
  END_VAR
  VAR_OUTPUT
    FreigabeHeizregisterOut : BOOL;  (* Freigabe an Heizregister *)
    DrehzahlHeizregisterOut : REAL;  (* ausgegebene Drehzahl Heizungspumpe *)
    FehlerOut : BOOL;  (* gespeicherter Fehler *)
  END_VAR

IF Freigabe THEN

    //Fehlerquittierung
    IF QuitFehler THEN
        FehlerOut := FALSE;
    END_IF;


    CASE uStep OF

        //AUS *********************************************************************************************
        0:
            IF stateEntry THEN
                stateEntry              := FALSE;
                FreigabeHeizregisterOut := FALSE;
                DrehzahlHeizregisterOut := 0.0;
            END_IF;

            //Automatikbetrieb aktiviert
            IF Automatikbetrieb AND NOT FehlerOut AND NOT FehlerSensorAussenluft THEN
                stateEntry := TRUE;
                uStep       := 1;
            ELSIF Dauerbetrieb AND NOT FehlerOut THEN
                stateEntry := TRUE;
                uStep       := 2;
            END_IF;


        //AUTOMATIKBETRIEB ********************************************************************************
        1:
            IF stateEntry THEN
                stateEntry := FALSE;
            END_IF;

            //Bei Neustart (Wetter nicht gut oder schlecht) ohne Verzögerung umschalten
            IF NOT loc_WetterIstSchlecht AND NOT loc_WetterIstGut THEN
                IF (FrischluftSattDefizitIst < FrischluftSattDefizitSoll) THEN
                    loc_WetterIstSchlecht := TRUE;
                ELSIF (FrischluftSattDefizitIst >= FrischluftSattDefizitSoll) THEN
                    loc_WetterIstGut := TRUE;
                END_IF;
            END_IF;

            //Umschaltverzögerung gutes Wetter / schlechtes Wetter
            TON_WetterIstGut(IN := loc_WetterIstSchlecht AND (FrischluftSattDefizitIst >= (FrischluftSattDefizitSoll + Hysterese)), PT := UmschaltverzWitterung);
            TON_WetterIstSchlecht(IN := loc_WetterIstGut AND (FrischluftSattDefizitIst < (FrischluftSattDefizitSoll - Hysterese)), PT := UmschaltverzWitterung);

            //Flankenauswertung (ersetzt EDGEPOS)
            R_TRIG_WetterIstGut(CLK := TON_WetterIstGut.Q);
            R_TRIG_WetterIstSchlecht(CLK := TON_WetterIstSchlecht.Q);

            IF R_TRIG_WetterIstGut.Q THEN
                loc_WetterIstGut      := TRUE;
                loc_WetterIstSchlecht := FALSE;
            ELSIF R_TRIG_WetterIstSchlecht.Q THEN
                loc_WetterIstGut      := FALSE;
                loc_WetterIstSchlecht := TRUE;
            END_IF;

            //Freigabe Heizregister
            FreigabeHeizregisterOut := loc_WetterIstSchlecht OR WetterIstSchlecht;
            DrehzahlHeizregisterOut := DrehzahlHeizregisterSoll;

            //Fehler
            IF FehlerSensorAussenluft THEN
                FehlerOut  := TRUE;
                stateEntry := TRUE;
                uStep       := 0;
            //Dauerbetrieb aktiv
            ELSIF Dauerbetrieb THEN
                stateEntry := TRUE;
                uStep       := 2;
            //Kein Automatikbetrieb
            ELSIF NOT Automatikbetrieb THEN
                stateEntry := TRUE;
                uStep       := 0;
            END_IF;


        //DAUERBETRIEB ***********************************************************************************
        2:
            IF stateEntry THEN
                stateEntry := FALSE;
            END_IF;

            //Freigabe Heizregister
            FreigabeHeizregisterOut := TRUE;
            DrehzahlHeizregisterOut := DrehzahlHeizregisterSoll;

            //Automatikbetrieb aktiv
            IF Automatikbetrieb THEN
                stateEntry := TRUE;
                uStep       := 1;
            //Kein Dauerbetrieb
            ELSIF NOT Dauerbetrieb THEN
                stateEntry := TRUE;
                uStep       := 0;
            END_IF;

    END_CASE;


ELSE

    FreigabeHeizregisterOut := FALSE;
    DrehzahlHeizregisterOut := 0.0;
    uStep                    := 0;
    stateEntry              := TRUE;
    FehlerOut               := FALSE;

END_IF;
END_FUNCTION_BLOCK

FUNCTION_BLOCK fbMathLuft
  VAR
    loc_Taupunkttemp : REAL;
    loc_TempK : REAL;  (* absolute Temperatur [K] *)
    loc_Nenner : REAL;  (* Magnus-Nenner (237.3 + T) *)
    loc_Basis : REAL;  (* Basis der Barometerformel *)
    loc_rF : REAL;  (* begrenzte rel. Feuchte [%] *)
  END_VAR
  VAR CONSTANT
    CONST_MATH_MAX_VALUE : REAL := 3.4e+38;
    CONST_MATH_DRUCK_MEERESHOEHE : REAL := 1013.25;
    C_LN10 : REAL := 2.30259;
  END_VAR
  VAR_INPUT
    Freigabe : BOOL;
    LuftTemperatur : REAL;  (* [°C] *)
    LuftRelFeuchte : REAL;  (* [%] *)
    MeterUeberAdria : REAL;  (* [m] *)
  END_VAR
  VAR_OUTPUT
    LuftAbsoluteFeuchteSatt : REAL;  (* [g/m³] *)
    LuftAbsoluteFeuchte_g_m3 : REAL;  (* [g/m³] *)
    LuftAbsoluteFeuchte_g_kg : REAL;  (* [g/kg] *)
    LuftSaettigungsdefizit : REAL;  (* [g/m³] *)
    LuftdruckUmgebung : REAL;  (* [hPa] *)
    LuftDichte : REAL;  (* [kg/m³] *)
    LuftDampfdruckSatt : REAL;  (* [mbar] *)
    LuftDampfdruckH2O : REAL;  (* [mbar] *)
    TaupunktTemp : REAL;  (* [°C] *)
    Gueltig : BOOL;  (* NEU: TRUE = alle Werte plausibel *)
  END_VAR

IF Freigabe THEN

	Gueltig    := TRUE;
	loc_TempK  := 273.15 + LuftTemperatur;
	loc_Nenner := 237.3  + LuftTemperatur;

	(* rel. Feuchte hart begrenzen - Sensorausreisser sonst durchgereicht *)
	loc_rF := LuftRelFeuchte;
	IF loc_rF < 0.0   THEN loc_rF := 0.0;   END_IF;
	IF loc_rF > 100.0 THEN loc_rF := 100.0; END_IF;


	(* --- Luftdruck [hPa] ------------------------------------------- *)
	(* p = p0 * (1 - 0.0065*h/288.15)^5.255                            *)
	loc_Basis := 1.0 - 0.0065 * MeterUeberAdria / 288.15;
	IF loc_Basis > 0.001 THEN
		LuftdruckUmgebung := CONST_MATH_DRUCK_MEERESHOEHE
		                     * EXP(5.255 * LN(loc_Basis));
	ELSE
		LuftdruckUmgebung := CONST_MATH_MAX_VALUE;
		Gueltig           := FALSE;
	END_IF;


	(* --- Luftdichte [kg/m³] ---------------------------------------- *)
	IF (loc_TempK > 0.001) AND (LuftdruckUmgebung < CONST_MATH_MAX_VALUE) THEN
		LuftDichte := (LuftdruckUmgebung * 100.0) / (287.058 * loc_TempK);
	ELSE
		LuftDichte := CONST_MATH_MAX_VALUE;
		Gueltig    := FALSE;
	END_IF;


	(* --- Saettigungsdampfdruck [mbar] ------------------------------ *)
	(* Magnus: es = 6.1078 * 10^(7.5*T/(237.3+T))                      *)
	IF loc_Nenner > 0.001 THEN
		LuftDampfdruckSatt := 6.1078
		                      * EXP(C_LN10 * 7.5 * LuftTemperatur / loc_Nenner);
	ELSE
		LuftDampfdruckSatt := CONST_MATH_MAX_VALUE;
		Gueltig            := FALSE;
	END_IF;


	(* --- Wasserdampfdruck [mbar] ----------------------------------- *)
	IF LuftDampfdruckSatt < CONST_MATH_MAX_VALUE THEN
		LuftDampfdruckH2O := LuftDampfdruckSatt * (loc_rF / 100.0);
	ELSE
		LuftDampfdruckH2O := CONST_MATH_MAX_VALUE;
		Gueltig           := FALSE;
	END_IF;


	(* --- absolute Feuchte gesaettigt [g/m³] ------------------------ *)
	IF (LuftDampfdruckSatt < CONST_MATH_MAX_VALUE) AND (loc_TempK > 0.001) THEN
		LuftAbsoluteFeuchteSatt := 216.67 * LuftDampfdruckSatt / loc_TempK;
	ELSE
		LuftAbsoluteFeuchteSatt := CONST_MATH_MAX_VALUE;
		Gueltig                 := FALSE;
	END_IF;


	(* --- absolute Feuchte [g/m³] ----------------------------------- *)
	IF LuftAbsoluteFeuchteSatt < CONST_MATH_MAX_VALUE THEN
		LuftAbsoluteFeuchte_g_m3 := (loc_rF / 100.0) * LuftAbsoluteFeuchteSatt;
	ELSE
		LuftAbsoluteFeuchte_g_m3 := CONST_MATH_MAX_VALUE;
		Gueltig                  := FALSE;
	END_IF;


	(* --- Saettigungsdefizit [g/m³] --------------------------------- *)
	IF LuftAbsoluteFeuchte_g_m3 < CONST_MATH_MAX_VALUE THEN
		LuftSaettigungsdefizit := LuftAbsoluteFeuchteSatt - LuftAbsoluteFeuchte_g_m3;
	ELSE
		LuftSaettigungsdefizit := CONST_MATH_MAX_VALUE;
		Gueltig                := FALSE;
	END_IF;


	(* --- absolute Feuchte [g/kg] ----------------------------------- *)
	IF (LuftAbsoluteFeuchte_g_m3 < CONST_MATH_MAX_VALUE)
	   AND (LuftDichte < CONST_MATH_MAX_VALUE) AND (LuftDichte > 0.001) THEN
		LuftAbsoluteFeuchte_g_kg := LuftAbsoluteFeuchte_g_m3 / LuftDichte;
	ELSE
		LuftAbsoluteFeuchte_g_kg := CONST_MATH_MAX_VALUE;
		Gueltig                  := FALSE;
	END_IF;


	(* --- Taupunkttemperatur [°C] ----------------------------------- *)
	IF (LuftDampfdruckH2O < CONST_MATH_MAX_VALUE) AND (LuftDampfdruckH2O > 0.001) THEN
		loc_Taupunkttemp := LN(LuftDampfdruckH2O) / C_LN10;   (* log10 *)
		IF (8.233 - loc_Taupunkttemp) > 0.001 THEN
			TaupunktTemp := (234.67 * loc_Taupunkttemp - 184.2)
			                / (8.233 - loc_Taupunkttemp);
		ELSE
			TaupunktTemp := CONST_MATH_MAX_VALUE;
			Gueltig      := FALSE;
		END_IF;
	ELSE
		TaupunktTemp := CONST_MATH_MAX_VALUE;
		Gueltig      := FALSE;
	END_IF;

ELSE

	LuftdruckUmgebung        := CONST_MATH_MAX_VALUE;
	LuftAbsoluteFeuchteSatt  := CONST_MATH_MAX_VALUE;
	LuftAbsoluteFeuchte_g_kg := CONST_MATH_MAX_VALUE;
	LuftAbsoluteFeuchte_g_m3 := CONST_MATH_MAX_VALUE;
	LuftDichte               := CONST_MATH_MAX_VALUE;
	TaupunktTemp             := CONST_MATH_MAX_VALUE;
	LuftDampfdruckH2O        := CONST_MATH_MAX_VALUE;
	LuftDampfdruckSatt       := CONST_MATH_MAX_VALUE;
	LuftSaettigungsdefizit   := CONST_MATH_MAX_VALUE;
	Gueltig                  := FALSE;

END_IF;
END_FUNCTION_BLOCK

FUNCTION_BLOCK fbCControlWitterung
  VAR
    i : USINT;
    SaettigungsdefizitIst : REAL;
    loc_WetterIstGut : BOOL;
    loc_WetterIstSchlecht : BOOL;
    TON_SchrittWitterung : TON;
    curStep : USINT;
    stateEntry : BOOL;
  END_VAR
  VAR_INPUT
    Freigabe : BOOL;
    MaterialfeuchteIst : UDINT;
    MaterialfeuchteStufe : ARRAY[1..6] OF UDINT;  (* absteigend! *)
    FrischluftSaettigungsdefizit : REAL;
    TrockenluftSaettigungsdefizit : REAL;
    AuswahlSensor : USINT;  (* 0=None 1=Frisch 2=Trocken *)
    SensorFrischluftVhd : BOOL;
    SensorTrockenluftVhd : BOOL;
    GrenzwertStufeAktuell : REAL;
    HystereseGrenzwert : REAL;
    VerzWetterwechsel : UDINT;  (* [ms] *)
    SchlechtwetterPulszeitAktuell : UDINT;
    SchlechtwetterPausezeitAktuell : UDINT;
  END_VAR
  VAR_OUTPUT
    StufeAktuell : USINT;
    WetterIstGut : BOOL;
    WetterIstSchlecht : BOOL;
    SchlechtwetterPulszeit : UDINT;
    SchlechtwetterPausezeit : UDINT;
    SensorGueltig : BOOL;  (* NEU - siehe Anmerkung 1 *)
  END_VAR

(********************************************************************
 * fbCControlWitterung - Portierung für EcoStruxure Machine Expert - HVAC
 ********************************************************************
 * Generierung der Witterungsverhaeltnisse aus Saettigungsdefizit
 * und Trocknungslaufzeit (Materialfeuchte-Stufe)
 ********************************************************************)
 
 IF Freigabe THEN

	(* --- Aktuell gueltige Stufe aus der Trockengutfeuchte ---------- *)
	(* Setzt eine ABSTEIGEND sortierte Schwellwerttabelle voraus!      *)
	StufeAktuell := 1;
	IF MaterialfeuchteIst <> 0 THEN
		FOR i := 1 TO 5 DO
			IF MaterialfeuchteIst <= MaterialfeuchteStufe[i] THEN
				StufeAktuell := i + 1;
			END_IF;
		END_FOR;
	END_IF;


	(* --- Puls-/Pausezeiten durchreichen ---------------------------- *)
	SchlechtwetterPulszeit  := SchlechtwetterPulszeitAktuell;
	SchlechtwetterPausezeit := SchlechtwetterPausezeitAktuell;


	(* --- Gueltigen Sensor bestimmen -------------------------------- *)
	SensorGueltig := TRUE;

	IF (AuswahlSensor = 1) AND SensorFrischluftVhd THEN
		SaettigungsdefizitIst := FrischluftSaettigungsdefizit;
	ELSIF (AuswahlSensor = 2) AND SensorTrockenluftVhd THEN
		SaettigungsdefizitIst := TrockenluftSaettigungsdefizit;
	(* Ausgewaehlter Sensor nicht vhd. -> Ersatzsensor in fester Reihenfolge *)
	ELSIF SensorFrischluftVhd THEN
		SaettigungsdefizitIst := FrischluftSaettigungsdefizit;
	ELSIF SensorTrockenluftVhd THEN
		SaettigungsdefizitIst := TrockenluftSaettigungsdefizit;
	ELSE
		SaettigungsdefizitIst := 0.0;
		SensorGueltig         := FALSE;   (* kein Sensor verfuegbar *)
	END_IF;


	(* --- Witterungsverhaeltnisse bestimmen ------------------------- *)
	IF SensorGueltig THEN

		loc_WetterIstGut      := FALSE;
		loc_WetterIstSchlecht := FALSE;

		IF SaettigungsdefizitIst >= (GrenzwertStufeAktuell + HystereseGrenzwert) THEN
			loc_WetterIstGut := TRUE;
		ELSIF SaettigungsdefizitIst <= (GrenzwertStufeAktuell - HystereseGrenzwert) THEN
			loc_WetterIstSchlecht := TRUE;
		END_IF;

		CASE curStep OF

		(* --- INIT --- *)
		0:
			TON_SchrittWitterung(IN := FALSE);
			stateEntry := TRUE;
			IF loc_WetterIstGut THEN
				curStep := 1;
			ELSE
				curStep := 2;
			END_IF;

		(* --- Wetter ist gut --- *)
		1:
			IF stateEntry THEN
				stateEntry := FALSE;
				TON_SchrittWitterung(IN := FALSE);
			END_IF;

			WetterIstGut      := TRUE;
			WetterIstSchlecht := FALSE;

			TON_SchrittWitterung(IN := loc_WetterIstSchlecht,
			                     PT := VerzWetterwechsel);

			IF TON_SchrittWitterung.Q THEN
				stateEntry := TRUE;
				curStep    := 2;
			END_IF;

		(* --- Wetter ist schlecht --- *)
		2:
			IF stateEntry THEN
				stateEntry := FALSE;
				TON_SchrittWitterung(IN := FALSE);
			END_IF;

			WetterIstGut      := FALSE;
			WetterIstSchlecht := TRUE;

			TON_SchrittWitterung(IN := loc_WetterIstGut,
			                     PT := VerzWetterwechsel);

			IF TON_SchrittWitterung.Q THEN
				stateEntry := TRUE;
				curStep    := 1;
			END_IF;

		ELSE
			curStep    := 0;      (* Schrittkette defensiv zuruecksetzen *)
			stateEntry := TRUE;

		END_CASE;

	ELSE
		(* Kein gueltiger Sensor -> Normalbetrieb, kein Schlechtwetter *)
		loc_WetterIstGut      := FALSE;
		loc_WetterIstSchlecht := FALSE;
		WetterIstGut          := TRUE;
		WetterIstSchlecht     := FALSE;
		TON_SchrittWitterung(IN := FALSE);
		stateEntry := TRUE;
		curStep    := 0;
	END_IF;


(* --- keine Freigabe des Bausteins --------------------------------- *)
ELSE
	loc_WetterIstGut        := FALSE;
	loc_WetterIstSchlecht   := FALSE;
	WetterIstGut            := FALSE;
	WetterIstSchlecht       := FALSE;
	SensorGueltig           := FALSE;
	TON_SchrittWitterung(IN := FALSE);
	stateEntry              := TRUE;
	curStep                 := 0;
	SaettigungsdefizitIst   := 0.0;
	SchlechtwetterPulszeit  := 0;
	SchlechtwetterPausezeit := 0;
	StufeAktuell            := 1;
END_IF;
 
END_FUNCTION_BLOCK

FUNCTION_BLOCK fbPulsPause
  VAR
    curStep : USINT;
    stateEntry : BOOL;
    TON_PulsPause : TON;
    loc_ET_ms : UDINT;
  END_VAR
  VAR_INPUT
    Freigabe : BOOL;  (* TRUE = Puls-/Pausebetrieb laeuft *)
    StartMitPause : BOOL;  (* Einstieg in die Pause statt Puls *)
    ZeitPuls : UDINT;  (* [ms] Trocknungszeit *)
    ZeitPause : UDINT;  (* [ms] Pausezeit, 0 = Dauerbetrieb *)
  END_VAR
  VAR_OUTPUT
    PulsOut : BOOL;  (* TRUE = jetzt trocknen *)
    PauseOut : BOOL;  (* TRUE = jetzt pausieren *)
    RestzeitPuls : UDINT;  (* [ms] *)
    RestzeitPause : UDINT;  (* [ms] *)
  END_VAR

IF Freigabe THEN

	(* --- Sonderfaelle ohne Schrittkette ---------------------------- *)
	IF ZeitPause = 0 THEN
		(* keine Pause parametriert -> durchgehend trocknen *)
		PulsOut       := TRUE;
		PauseOut      := FALSE;
		RestzeitPuls  := ZeitPuls;
		RestzeitPause := 0;
		TON_PulsPause(IN := FALSE, PT := 0);
		curStep       := 0;
		stateEntry    := TRUE;

	ELSIF ZeitPuls = 0 THEN
		(* keine Laufzeit parametriert -> Box bleibt aus *)
		PulsOut       := FALSE;
		PauseOut      := TRUE;
		RestzeitPuls  := 0;
		RestzeitPause := ZeitPause;
		TON_PulsPause(IN := FALSE, PT := 0);
		curStep       := 0;
		stateEntry    := TRUE;

	ELSE

		CASE curStep OF

		(* --- INIT --- *)
		0:
			TON_PulsPause(IN := FALSE, PT := 0);
			stateEntry := TRUE;
			IF StartMitPause THEN
				curStep := 2;
			ELSE
				curStep := 1;
			END_IF;

		(* --- PULS: Box trocknet --- *)
		1:
			IF stateEntry THEN
				stateEntry := FALSE;
				TON_PulsPause(IN := FALSE, PT := 0);
			END_IF;

			PulsOut  := TRUE;
			PauseOut := FALSE;

			TON_PulsPause(IN := TRUE, PT := ZeitPuls);

			IF TON_PulsPause.Q THEN
				stateEntry := TRUE;
				curStep    := 2;
			END_IF;

		(* --- PAUSE: Box steht --- *)
		2:
			IF stateEntry THEN
				stateEntry := FALSE;
				TON_PulsPause(IN := FALSE, PT := 0);
			END_IF;

			PulsOut  := FALSE;
			PauseOut := TRUE;

			TON_PulsPause(IN := TRUE, PT := ZeitPause);

			IF TON_PulsPause.Q THEN
				stateEntry := TRUE;
				curStep    := 1;
			END_IF;

		ELSE
			curStep    := 0;
			stateEntry := TRUE;

		END_CASE;


		(* --- Restzeiten fuer die HMI-Anzeige --- *)
		IF stateEntry THEN
			(* Schrittwechsel: Timer wird erst im naechsten Zyklus gestartet *)
			RestzeitPuls  := ZeitPuls;
			RestzeitPause := ZeitPause;
		ELSE
			loc_ET_ms := TON_PulsPause.ET;

